LIN {X 99.425,Y -44.827,Z -45.204,A -90.000,B 90.000,C 0.000} C_DIS
LIN {X 99.466,Y -44.816,Z -45.164,A -90.000,B 90.000,C 0.000} C_DIS
LIN {X 99.493,Y -44.805,Z -45.135,A -90.000,B 90.000,C 0.000} C_DIS
LIN {X 99.508,Y -44.792,Z -45.118,A -90.000,B 90.000,C 0.000} C_DIS
LIN {X 99.515,Y -44.777,Z -45.107,A -90.000,B 90.000,C 0.000} C_DIS
LIN {X 99.516,Y -44.768,Z -45.104,A -90.000,B 90.000,C 0.000} C_DIS
LIN {X 99.507,Y -44.687,Z -45.089,A -90.000,B 90.000,C 0.000} C_DIS
LIN {X 99.509,Y -44.621,Z -45.070,A -90.000,B 90.000,C 0.000} C_DIS
LIN {X 99.519,Y -44.564,Z -45.046,A -90.000,B 90.000,C 0.000} C_DIS
LIN {X 99.538,Y -44.495,Z -45.011,A -90.000,B 90.000,C 0.000} C_DIS
LIN {X 99.570,Y -44.412,Z -44.962,A -90.000,B 90.000,C 0.000} C_DIS
LIN {X 99.618,Y -44.314,Z -44.895,A -90.000,B 90.000,C 0.000} C_DIS
LIN {X 99.683,Y -44.199,Z -44.808,A -90.000,B 90.000,C 0.000} C_DIS
LIN {X 99.768,Y -44.065,Z -44.699,A -90.000,B 90.000,C 0.000} C_DIS
LIN {X 99.877,Y -43.910,Z -44.564,A -90.000,B 90.000,C 0.000} C_DIS
LIN {X 100.012,Y -43.731,Z -44.402,A -90.000,B 90.000,C 0.000} C_DIS
LIN {X 100.175,Y -43.526,Z -44.208,A -90.000,B 90.000,C 0.000} C_DIS
LIN {X 100.317,Y -43.354,Z -44.041,A -90.000,B 90.000,C 0.000} C_DIS
LIN {X 100.597,Y -43.062,Z -43.718,A -90.000,B 90.000,C 0.000} C_DIS
LIN {X 100.862,Y -42.817,Z -43.416,A -90.000,B 90.000,C 0.000} C_DIS
LIN {X 101.165,Y -37.308,Z -43.072,A -90.000,B 90.000,C 0.000} C_DIS
LIN {X 101.207,Y -37.308,Z -43.025,A -90.000,B 90.000,C 0.000} C_DIS
LIN {X 101.288,Y -42.488,Z -42.934,A -90.000,B 90.000,C 0.000} C_DIS
LIN {X 101.299,Y -42.484,Z -42.922,A -90.000,B 90.000,C 0.000} C_DIS
LIN {X 101.301,Y -42.492,Z -42.920,A -90.000,B 90.000,C 0.000} C_DIS
LIN {X 101.311,Y -42.494,Z -42.909,A -90.000,B 90.000,C 0.000} C_DIS
LIN {X 101.393,Y -37.308,Z -42.819,A -90.000,B 90.000,C 0.000} C_DIS
LIN {X 101.467,Y -37.311,Z -42.737,A -90.000,B 90.000,C 0.000} C_DIS
LIN {X 101.519,Y -37.308,Z -42.679,A -90.000,B 90.000,C 0.000} C_DIS
LIN {X 101.519,Y -60.000,Z -42.679,A -90.000,B 90.000,C 0.000} C_DIS
LIN {X 91.034,Y -60.000,Z -118.889,A -90.000,B 90.000,C 0.000} C_DIS
LIN {X 91.034,Y -37.308,Z -118.889,A -90.000,B 90.000,C 0.000} C_DIS
LIN {X 91.028,Y -37.310,Z -119.075,A -90.000,B 90.000,C 0.000} C_DIS
LIN {X 91.024,Y -37.317,Z -119.386,A -90.000,B 90.000,C 0.000} C_DIS
LIN {X 91.058,Y -37.308,Z -120.562,A -90.000,B 90.000,C 0.000} C_DIS
LIN {X 91.058,Y -60.000,Z -120.562,A -90.000,B 90.000,C 0.000} C_DIS
LIN {X 18.246,Y -60.000,Z -172.708,A -90.000,B 90.000,C 0.000} C_DIS
LIN {X 18.246,Y -37.308,Z -172.708,A -90.000,B 90.000,C 0.000} C_DIS
LIN {X 18.676,Y -37.337,Z -172.279,A -90.000,B 90.000,C 0.000} C_DIS
LIN {X 19.234,Y -37.370,Z -171.709,A -90.000,B 90.000,C 0.000} C_DIS
LIN {X 19.511,Y -37.385,Z -171.418,A -90.000,B 90.000,C 0.000} C_DIS
LIN {X 20.129,Y -37.438,Z -170.757,A -90.000,B 90.000,C 0.000} C_DIS
LIN {X 20.879,Y -37.487,Z -169.898,A -90.000,B 90.000,C 0.000} C_DIS
LIN {X 21.061,Y -37.497,Z -169.689,A -90.000,B 90.000,C 0.000} C_DIS
LIN {X 21.262,Y -37.507,Z -169.454,A -90.000,B 90.000,C 0.000} C_DIS
LIN {X 21.665,Y -37.542,Z -168.973,A -90.000,B 90.000,C 0.000} C_DIS
LIN {X 21.886,Y -37.558,Z -168.693,A -90.000,B 90.000,C 0.000} C_DIS
LIN {X 22.441,Y -37.593,Z -167.976,A -90.000,B 90.000,C 0.000} C_DIS
LIN {X 22.927,Y -37.634,Z -167.341,A -90.000,B 90.000,C 0.000} C_DIS
LIN {X 23.381,Y -37.667,Z -166.718,A -90.000,B 90.000,C 0.000} C_DIS
LIN {X 23.591,Y -37.681,Z -166.424,A -90.000,B 90.000,C 0.000} C_DIS
LIN {X 23.790,Y -37.709,Z -166.136,A -90.000,B 90.000,C 0.000} C_DIS
LIN {X 23.902,Y -37.722,Z -165.976,A -90.000,B 90.000,C 0.000} C_DIS
LIN {X 24.323,Y -37.756,Z -165.386,A -90.000,B 90.000,C 0.000} C_DIS
LIN {X 24.729,Y -37.786,Z -164.795,A -90.000,B 90.000,C 0.000} C_DIS
LIN {X 25.418,Y -37.885,Z -163.750,A -90.000,B 90.000,C 0.000} C_DIS
LIN {X 25.616,Y -37.899,Z -163.459,A -90.000,B 90.000,C 0.000} C_DIS
LIN {X 25.783,Y -37.929,Z -163.201,A -90.000,B 90.000,C 0.000} C_DIS
LIN {X 26.867,Y -38.118,Z -161.513,A -90.000,B 90.000,C 0.000} C_DIS
LIN {X 26.926,Y -38.131,Z -161.421,A -90.000,B 90.000,C 0.000} C_DIS
LIN {X 27.075,Y -38.162,Z -161.189,A -90.000,B 90.000,C 0.000} C_DIS
LIN {X 27.785,Y -38.314,Z -160.034,A -90.000,B 90.000,C 0.000} C_DIS
LIN {X 28.223,Y -38.430,Z -159.320,A -90.000,B 90.000,C 0.000} C_DIS
LIN {X 28.758,Y -38.583,Z -158.366,A -90.000,B 90.000,C 0.000} C_DIS
LIN {X 29.089,Y -38.675,Z -157.778,A -90.000,B 90.000,C 0.000} C_DIS
LIN {X 28.763,Y -38.667,Z -157.817,A -90.000,B 90.000,C 0.000} C_DIS
LIN {X 28.657,Y -38.665,Z -157.825,A -90.000,B 90.000,C 0.000} C_DIS
LIN {X 28.540,Y -38.663,Z -157.832,A -90.000,B 90.000,C 0.000} C_DIS
LIN {X 28.360,Y -38.661,Z -157.834,A -90.000,B 90.000,C 0.000} C_DIS
LIN {X 28.193,Y -38.664,Z -157.832,A -90.000,B 90.000,C 0.000} C_DIS
LIN {X 27.973,Y -38.669,Z -157.816,A -90.000,B 90.000,C 0.000} C_DIS
LIN {X 27.602,Y -38.679,Z -157.774,A -90.000,B 90.000,C 0.000} C_DIS
LIN {X 27.471,Y -38.683,Z -157.755,A -90.000,B 90.000,C 0.000} C_DIS
LIN {X 27.348,Y -38.686,Z -157.733,A -90.000,B 90.000,C 0.000} C_DIS
LIN {X 27.168,Y -38.691,Z -157.696,A -90.000,B 90.000,C 0.000} C_DIS
LIN {X 26.963,Y -38.699,Z -157.642,A -90.000,B 90.000,C 0.000} C_DIS
LIN {X 26.817,Y -38.705,Z -157.597,A -90.000,B 90.000,C 0.000} C_DIS
LIN {X 26.706,Y -38.710,Z -157.559,A -90.000,B 90.000,C 0.000} C_DIS
LIN {X 26.470,Y -38.713,Z -157.462,A -90.000,B 90.000,C 0.000} C_DIS
LIN {X 26.304,Y -38.715,Z -157.392,A -90.000,B 90.000,C 0.000} C_DIS
LIN {X 26.199,Y -38.718,Z -157.343,A -90.000,B 90.000,C 0.000} C_DIS
LIN {X 26.036,Y -38.724,Z -157.251,A -90.000,B 90.000,C 0.000} C_DIS
LIN {X 25.598,Y -38.746,Z -156.984,A -90.000,B 90.000,C 0.000} C_DIS
LIN {X 25.482,Y -38.751,Z -156.901,A -90.000,B 90.000,C 0.000} C_DIS
LIN {X 25.247,Y -38.759,Z -156.714,A -90.000,B 90.000,C 0.000} C_DIS
LIN {X 25.138,Y -38.762,Z -156.620,A -90.000,B 90.000,C 0.000} C_DIS
LIN {X 25.035,Y -38.762,Z -156.525,A -90.000,B 90.000,C 0.000} C_DIS
LIN {X 24.917,Y -38.757,Z -156.404,A -90.000,B 90.000,C 0.000} C_DIS
LIN {X 24.794,Y -38.750,Z -156.269,A -90.000,B 90.000,C 0.000} C_DIS
LIN {X 24.611,Y -38.747,Z -156.042,A -90.000,B 90.000,C 0.000} C_DIS
LIN {X 24.050,Y -38.739,Z -155.340,A -90.000,B 90.000,C 0.000} C_DIS
LIN {X 23.907,Y -38.734,Z -155.160,A -90.000,B 90.000,C 0.000} C_DIS
LIN {X 23.791,Y -38.721,Z -155.008,A -90.000,B 90.000,C 0.000} C_DIS
LIN {X 23.677,Y -38.702,Z -154.847,A -90.000,B 90.000,C 0.000} C_DIS
LIN {X 23.524,Y -38.677,Z -154.617,A -90.000,B 90.000,C 0.000} C_DIS
LIN {X 23.421,Y -38.661,Z -154.444,A -90.000,B 90.000,C 0.000} C_DIS
LIN {X 23.386,Y -38.655,Z -154.380,A -90.000,B 90.000,C 0.000} C_DIS
LIN {X 23.328,Y -38.647,Z -154.260,A -90.000,B 90.000,C 0.000} C_DIS
LIN {X 23.170,Y -38.626,Z -153.901,A -90.000,B 90.000,C 0.000} C_DIS
LIN {X 23.071,Y -38.615,Z -153.627,A -90.000,B 90.000,C 0.000} C_DIS
LIN {X 23.025,Y -38.608,Z -153.480,A -90.000,B 90.000,C 0.000} C_DIS
LIN {X 23.006,Y -38.602,Z -153.415,A -90.000,B 90.000,C 0.000} C_DIS
LIN {X 22.974,Y -38.590,Z -153.292,A -90.000,B 90.000,C 0.000} C_DIS
LIN {X 22.949,Y -38.580,Z -153.182,A -90.000,B 90.000,C 0.000} C_DIS
LIN {X 22.929,Y -38.570,Z -153.079,A -90.000,B 90.000,C 0.000} C_DIS
LIN {X 22.906,Y -38.558,Z -152.910,A -90.000,B 90.000,C 0.000} C_DIS
LIN {X 22.877,Y -38.535,Z -152.666,A -90.000,B 90.000,C 0.000} C_DIS
LIN {X 22.866,Y -38.520,Z -152.493,A -90.000,B 90.000,C 0.000} C_DIS
LIN {X 22.858,Y -38.505,Z -152.287,A -90.000,B 90.000,C 0.000} C_DIS
LIN {X 22.857,Y -38.492,Z -152.102,A -90.000,B 90.000,C 0.000} C_DIS
LIN {X 22.860,Y -38.479,Z -151.897,A -90.000,B 90.000,C 0.000} C_DIS
LIN {X 22.879,Y -38.466,Z -151.654,A -90.000,B 90.000,C 0.000} C_DIS
LIN {X 22.890,Y -38.460,Z -151.561,A -90.000,B 90.000,C 0.000} C_DIS
LIN {X 22.930,Y -38.448,Z -151.318,A -90.000,B 90.000,C 0.000} C_DIS
LIN {X 22.962,Y -38.439,Z -151.169,A -90.000,B 90.000,C 0.000} C_DIS
LIN {X 23.121,Y -38.404,Z -150.496,A -90.000,B 90.000,C 0.000} C_DIS
LIN {X 23.299,Y -38.353,Z -149.757,A -90.000,B 90.000,C 0.000} C_DIS
LIN {X 23.377,Y -38.318,Z -149.455,A -90.000,B 90.000,C 0.000} C_DIS
LIN {X 23.475,Y -38.278,Z -149.098,A -90.000,B 90.000,C 0.000} C_DIS
LIN {X 22.762,Y -38.124,Z -149.465,A -90.000,B 90.000,C 0.000} C_DIS
LIN {X 22.308,Y -38.024,Z -149.687,A -90.000,B 90.000,C 0.000} C_DIS
LIN {X 21.806,Y -37.911,Z -149.923,A -90.000,B 90.000,C 0.000} C_DIS
LIN {X 21.521,Y -37.843,Z -150.045,A -90.000,B 90.000,C 0.000} C_DIS
LIN {X 21.069,Y -37.732,Z -150.227,A -90.000,B 90.000,C 0.000} C_DIS
LIN {X 20.845,Y -37.674,Z -150.314,A -90.000,B 90.000,C 0.000} C_DIS
LIN {X 20.751,Y -37.647,Z -150.349,A -90.000,B 90.000,C 0.000} C_DIS
LIN {X 20.361,Y -37.529,Z -150.492,A -90.000,B 90.000,C 0.000} C_DIS
LIN {X 20.188,Y -37.475,Z -150.553,A -90.000,B 90.000,C 0.000} C_DIS
LIN {X 19.812,Y -37.357,Z -150.680,A -90.000,B 90.000,C 0.000} C_DIS
LIN {X 19.659,Y -37.308,Z -150.727,A -90.000,B 90.000,C 0.000} C_DIS
LIN {X 19.659,Y -60.000,Z -150.727,A -90.000,B 90.000,C 0.000} C_DIS
LIN {X 22.617,Y -60.000,Z -164.416,A -90.000,B 90.000,C 0.000} C_DIS
LIN {X 22.617,Y -37.308,Z -164.416,A -90.000,B 90.000,C 0.000} C_DIS
LIN {X 22.733,Y -37.343,Z -164.245,A -90.000,B 90.000,C 0.000} C_DIS
LIN {X 23.104,Y -37.453,Z -163.677,A -90.000,B 90.000,C 0.000} C_DIS
LIN {X 23.691,Y -37.627,Z -162.765,A -90.000,B 90.000,C 0.000} C_DIS
LIN {X 23.962,Y -37.712,Z -162.351,A -90.000,B 90.000,C 0.000} C_DIS
LIN {X 24.575,Y -37.908,Z -161.385,A -90.000,B 90.000,C 0.000} C_DIS
LIN {X 25.260,Y -38.149,Z -160.314,A -90.000,B 90.000,C 0.000} C_DIS
LIN {X 25.375,Y -38.189,Z -160.136,A -90.000,B 90.000,C 0.000} C_DIS
LIN {X 25.866,Y -38.354,Z -159.341,A -90.000,B 90.000,C 0.000} C_DIS
LIN {X 25.505,Y -38.359,Z -159.191,A -90.000,B 90.000,C 0.000} C_DIS
LIN {X 25.293,Y -38.363,Z -159.090,A -90.000,B 90.000,C 0.000} C_DIS
LIN {X 25.088,Y -38.371,Z -158.977,A -90.000,B 90.000,C 0.000} C_DIS
LIN {X 24.998,Y -38.375,Z -158.925,A -90.000,B 90.000,C 0.000} C_DIS
LIN {X 24.767,Y -38.384,Z -158.783,A -90.000,B 90.000,C 0.000} C_DIS
LIN {X 24.591,Y -38.384,Z -158.674,A -90.000,B 90.000,C 0.000} C_DIS
LIN {X 24.446,Y -38.384,Z -158.578,A -90.000,B 90.000,C 0.000} C_DIS
LIN {X 24.331,Y -38.386,Z -158.495,A -90.000,B 90.000,C 0.000} C_DIS
LIN {X 24.251,Y -38.388,Z -158.435,A -90.000,B 90.000,C 0.000} C_DIS
LIN {X 24.016,Y -38.394,Z -158.248,A -90.000,B 90.000,C 0.000} C_DIS
LIN {X 23.824,Y -38.401,Z -158.084,A -90.000,B 90.000,C 0.000} C_DIS
LIN {X 23.677,Y -38.403,Z -157.949,A -90.000,B 90.000,C 0.000} C_DIS
LIN {X 23.542,Y -38.396,Z -157.812,A -90.000,B 90.000,C 0.000} C_DIS
LIN {X 23.436,Y -38.389,Z -157.699,A -90.000,B 90.000,C 0.000} C_DIS
LIN {X 23.308,Y -38.381,Z -157.555,A -90.000,B 90.000,C 0.000} C_DIS
LIN {X 22.995,Y -38.364,Z -157.164,A -90.000,B 90.000,C 0.000} C_DIS
LIN {X 22.933,Y -38.361,Z -157.086,A -90.000,B 90.000,C 0.000} C_DIS
LIN {X 22.850,Y -38.356,Z -156.982,A -90.000,B 90.000,C 0.000} C_DIS
LIN {X 22.614,Y -38.352,Z -156.685,A -90.000,B 90.000,C 0.000} C_DIS
LIN {X 22.511,Y -38.348,Z -156.555,A -90.000,B 90.000,C 0.000} C_DIS
LIN {X 22.379,Y -38.333,Z -156.386,A -90.000,B 90.000,C 0.000} C_DIS
LIN {X 22.216,Y -38.305,Z -156.169,A -90.000,B 90.000,C 0.000} C_DIS
LIN {X 22.071,Y -38.279,Z -155.962,A -90.000,B 90.000,C 0.000} C_DIS
LIN {X 21.887,Y -38.248,Z -155.683,A -90.000,B 90.000,C 0.000} C_DIS
LIN {X 21.768,Y -38.229,Z -155.484,A -90.000,B 90.000,C 0.000} C_DIS
LIN {X 21.691,Y -38.217,Z -155.345,A -90.000,B 90.000,C 0.000} C_DIS
LIN {X 21.617,Y -38.206,Z -155.200,A -90.000,B 90.000,C 0.000} C_DIS
LIN {X 21.556,Y -38.197,Z -155.070,A -90.000,B 90.000,C 0.000} C_DIS
LIN {X 21.488,Y -38.185,Z -154.914,A -90.000,B 90.000,C 0.000} C_DIS
LIN {X 21.411,Y -38.163,Z -154.732,A -90.000,B 90.000,C 0.000} C_DIS
LIN {X 21.349,Y -38.144,Z -154.572,A -90.000,B 90.000,C 0.000} C_DIS
LIN {X 21.232,Y -38.110,Z -154.231,A -90.000,B 90.000,C 0.000} C_DIS
LIN {X 21.148,Y -38.084,Z -153.946,A -90.000,B 90.000,C 0.000} C_DIS
LIN {X 21.104,Y -38.067,Z -153.773,A -90.000,B 90.000,C 0.000} C_DIS
LIN {X 21.062,Y -38.048,Z -153.578,A -90.000,B 90.000,C 0.000} C_DIS
LIN {X 21.032,Y -38.034,Z -153.418,A -90.000,B 90.000,C 0.000} C_DIS
LIN {X 20.994,Y -38.014,Z -153.140,A -90.000,B 90.000,C 0.000} C_DIS
LIN {X 20.968,Y -37.998,Z -152.925,A -90.000,B 90.000,C 0.000} C_DIS
LIN {X 20.955,Y -37.988,Z -152.775,A -90.000,B 90.000,C 0.000} C_DIS
LIN {X 20.945,Y -37.976,Z -152.609,A -90.000,B 90.000,C 0.000} C_DIS
LIN {X 20.936,Y -37.959,Z -152.359,A -90.000,B 90.000,C 0.000} C_DIS
LIN {X 20.612,Y -37.866,Z -152.471,A -90.000,B 90.000,C 0.000} C_DIS
LIN {X 20.258,Y -37.764,Z -152.587,A -90.000,B 90.000,C 0.000} C_DIS
LIN {X 20.104,Y -37.719,Z -152.633,A -90.000,B 90.000,C 0.000} C_DIS
LIN {X 19.527,Y -37.545,Z -152.708,A -90.000,B 90.000,C 0.000} C_DIS
LIN {X 19.410,Y -37.509,Z -152.701,A -90.000,B 90.000,C 0.000} C_DIS
LIN {X 19.315,Y -37.479,Z -152.689,A -90.000,B 90.000,C 0.000} C_DIS
LIN {X 19.266,Y -37.463,Z -152.682,A -90.000,B 90.000,C 0.000} C_DIS
LIN {X 19.149,Y -37.425,Z -152.657,A -90.000,B 90.000,C 0.000} C_DIS
LIN {X 19.091,Y -37.406,Z -152.642,A -90.000,B 90.000,C 0.000} C_DIS
LIN {X 18.945,Y -37.358,Z -152.594,A -90.000,B 90.000,C 0.000} C_DIS
LIN {X 18.894,Y -37.340,Z -152.574,A -90.000,B 90.000,C 0.000} C_DIS
LIN {X 18.810,Y -37.308,Z -152.537,A -90.000,B 90.000,C 0.000} C_DIS
LIN {X 18.810,Y -60.000,Z -152.537,A -90.000,B 90.000,C 0.000} C_DIS
LIN {X 21.484,Y -60.000,Z -162.510,A -90.000,B 90.000,C 0.000} C_DIS
LIN {X 21.484,Y -37.308,Z -162.510,A -90.000,B 90.000,C 0.000} C_DIS
LIN {X 21.876,Y -37.483,Z -161.895,A -90.000,B 90.000,C 0.000} C_DIS
LIN {X 22.026,Y -37.546,Z -161.659,A -90.000,B 90.000,C 0.000} C_DIS
LIN {X 22.297,Y -37.662,Z -161.243,A -90.000,B 90.000,C 0.000} C_DIS
LIN {X 23.082,Y -37.985,Z -160.008,A -90.000,B 90.000,C 0.000} C_DIS
LIN {X 22.787,Y -37.991,Z -159.774,A -90.000,B 90.000,C 0.000} C_DIS
LIN {X 22.571,Y -37.983,Z -159.586,A -90.000,B 90.000,C 0.000} C_DIS
LIN {X 22.497,Y -37.980,Z -159.520,A -90.000,B 90.000,C 0.000} C_DIS
LIN {X 22.296,Y -37.971,Z -159.329,A -90.000,B 90.000,C 0.000} C_DIS
LIN {X 22.236,Y -37.969,Z -159.269,A -90.000,B 90.000,C 0.000} C_DIS
LIN {X 22.077,Y -37.956,Z -159.103,A -90.000,B 90.000,C 0.000} C_DIS
LIN {X 21.980,Y -37.944,Z -158.996,A -90.000,B 90.000,C 0.000} C_DIS
LIN {X 21.844,Y -37.927,Z -158.840,A -90.000,B 90.000,C 0.000} C_DIS
LIN {X 21.720,Y -37.913,Z -158.684,A -90.000,B 90.000,C 0.000} C_DIS
LIN {X 21.264,Y -37.892,Z -158.113,A -90.000,B 90.000,C 0.000} C_DIS
LIN {X 21.115,Y -37.884,Z -157.924,A -90.000,B 90.000,C 0.000} C_DIS
LIN {X 20.990,Y -37.866,Z -157.761,A -90.000,B 90.000,C 0.000} C_DIS
LIN {X 20.835,Y -37.840,Z -157.559,A -90.000,B 90.000,C 0.000} C_DIS
LIN {X 20.635,Y -37.803,Z -157.287,A -90.000,B 90.000,C 0.000} C_DIS
LIN {X 20.482,Y -37.779,Z -157.068,A -90.000,B 90.000,C 0.000} C_DIS
LIN {X 20.297,Y -37.751,Z -156.789,A -90.000,B 90.000,C 0.000} C_DIS
LIN {X 20.213,Y -37.739,Z -156.654,A -90.000,B 90.000,C 0.000} C_DIS
LIN {X 20.089,Y -37.722,Z -156.444,A -90.000,B 90.000,C 0.000} C_DIS
LIN {X 19.980,Y -37.709,Z -156.249,A -90.000,B 90.000,C 0.000} C_DIS
LIN {X 19.867,Y -37.686,Z -156.016,A -90.000,B 90.000,C 0.000} C_DIS
LIN {X 19.744,Y -37.658,Z -155.740,A -90.000,B 90.000,C 0.000} C_DIS
LIN {X 19.635,Y -37.632,Z -155.484,A -90.000,B 90.000,C 0.000} C_DIS
LIN {X 19.572,Y -37.617,Z -155.324,A -90.000,B 90.000,C 0.000} C_DIS
LIN {X 19.541,Y -37.610,Z -155.241,A -90.000,B 90.000,C 0.000} C_DIS
LIN {X 19.422,Y -37.583,Z -154.899,A -90.000,B 90.000,C 0.000} C_DIS
LIN {X 19.361,Y -37.570,Z -154.701,A -90.000,B 90.000,C 0.000} C_DIS
LIN {X 19.198,Y -37.517,Z -154.690,A -90.000,B 90.000,C 0.000} C_DIS
LIN {X 19.005,Y -37.454,Z -154.665,A -90.000,B 90.000,C 0.000} C_DIS
LIN {X 18.852,Y -37.405,Z -154.637,A -90.000,B 90.000,C 0.000} C_DIS
LIN {X 18.741,Y -37.370,Z -154.614,A -90.000,B 90.000,C 0.000} C_DIS
LIN {X 18.608,Y -37.327,Z -154.581,A -90.000,B 90.000,C 0.000} C_DIS
LIN {X 18.552,Y -37.308,Z -154.565,A -90.000,B 90.000,C 0.000} C_DIS
LIN {X 18.417,Y -37.265,Z -154.530,A -90.000,B 90.000,C 0.000} C_DIS
LIN {X 18.286,Y -37.220,Z -154.499,A -90.000,B 90.000,C 0.000} C_DIS
LIN {X 18.158,Y -37.176,Z -154.474,A -90.000,B 90.000,C 0.000} C_DIS
LIN {X 18.033,Y -37.133,Z -154.454,A -90.000,B 90.000,C 0.000} C_DIS
LIN {X 17.913,Y -37.092,Z -154.438,A -90.000,B 90.000,C 0.000} C_DIS
LIN {X 17.796,Y -37.052,Z -154.428,A -90.000,B 90.000,C 0.000} C_DIS
LIN {X 17.682,Y -37.013,Z -154.422,A -90.000,B 90.000,C 0.000} C_DIS
LIN {X 17.518,Y -36.957,Z -154.423,A -90.000,B 90.000,C 0.000} C_DIS
LIN {X 17.413,Y -36.921,Z -154.429,A -90.000,B 90.000,C 0.000} C_DIS
LIN {X 17.311,Y -36.887,Z -154.439,A -90.000,B 90.000,C 0.000} C_DIS
LIN {X 17.213,Y -36.854,Z -154.454,A -90.000,B 90.000,C 0.000} C_DIS
LIN {X 17.072,Y -36.807,Z -154.485,A -90.000,B 90.000,C 0.000} C_DIS
LIN {X 16.982,Y -36.777,Z -154.510,A -90.000,B 90.000,C 0.000} C_DIS
LIN {X 16.896,Y -36.748,Z -154.539,A -90.000,B 90.000,C 0.000} C_DIS
LIN {X 16.812,Y -36.721,Z -154.573,A -90.000,B 90.000,C 0.000} C_DIS
LIN {X 16.693,Y -36.682,Z -154.630,A -90.000,B 90.000,C 0.000} C_DIS
LIN {X 16.618,Y -36.657,Z -154.673,A -90.000,B 90.000,C 0.000} C_DIS
LIN {X 16.545,Y -36.634,Z -154.719,A -90.000,B 90.000,C 0.000} C_DIS
LIN {X 16.476,Y -36.611,Z -154.769,A -90.000,B 90.000,C 0.000} C_DIS
LIN {X 16.378,Y -36.580,Z -154.851,A -90.000,B 90.000,C 0.000} C_DIS
LIN {X 16.316,Y -36.560,Z -154.909,A -90.000,B 90.000,C 0.000} C_DIS
LIN {X 16.229,Y -36.530,Z -155.003,A -90.000,B 90.000,C 0.000} C_DIS
LIN {X 16.175,Y -36.511,Z -155.069,A -90.000,B 90.000,C 0.000} C_DIS
LIN {X 16.099,Y -36.483,Z -155.174,A -90.000,B 90.000,C 0.000} C_DIS
LIN {X 16.007,Y -36.446,Z -155.323,A -90.000,B 90.000,C 0.000} C_DIS
LIN {X 15.965,Y -36.428,Z -155.402,A -90.000,B 90.000,C 0.000} C_DIS
LIN {X 15.891,Y -36.387,Z -155.567,A -90.000,B 90.000,C 0.000} C_DIS
LIN {X 15.826,Y -36.349,Z -155.742,A -90.000,B 90.000,C 0.000} C_DIS
LIN {X 15.798,Y -36.331,Z -155.833,A -90.000,B 90.000,C 0.000} C_DIS
LIN {X 15.750,Y -36.297,Z -156.020,A -90.000,B 90.000,C 0.000} C_DIS
LIN {X 15.712,Y -36.266,Z -156.215,A -90.000,B 90.000,C 0.000} C_DIS
LIN {X 15.683,Y -36.238,Z -156.416,A -90.000,B 90.000,C 0.000} C_DIS
LIN {X 15.664,Y -36.214,Z -156.624,A -90.000,B 90.000,C 0.000} C_DIS
LIN {X 15.655,Y -36.192,Z -156.837,A -90.000,B 90.000,C 0.000} C_DIS
LIN {X 15.654,Y -36.168,Z -157.055,A -90.000,B 90.000,C 0.000} C_DIS
LIN {X 15.663,Y -36.139,Z -157.276,A -90.000,B 90.000,C 0.000} C_DIS
LIN {X 15.670,Y -36.125,Z -157.388,A -90.000,B 90.000,C 0.000} C_DIS
LIN {X 15.691,Y -36.100,Z -157.613,A -90.000,B 90.000,C 0.000} C_DIS
LIN {X 15.721,Y -36.078,Z -157.841,A -90.000,B 90.000,C 0.000} C_DIS
LIN {X 15.758,Y -36.064,Z -158.069,A -90.000,B 90.000,C 0.000} C_DIS
LIN {X 15.803,Y -36.055,Z -158.298,A -90.000,B 90.000,C 0.000} C_DIS
LIN {X 15.856,Y -36.047,Z -158.527,A -90.000,B 90.000,C 0.000} C_DIS
LIN {X 15.916,Y -36.040,Z -158.754,A -90.000,B 90.000,C 0.000} C_DIS
LIN {X 15.982,Y -36.035,Z -158.980,A -90.000,B 90.000,C 0.000} C_DIS
LIN {X 16.056,Y -36.034,Z -159.203,A -90.000,B 90.000,C 0.000} C_DIS
LIN {X 16.135,Y -36.036,Z -159.423,A -90.000,B 90.000,C 0.000} C_DIS
LIN {X 16.221,Y -36.040,Z -159.638,A -90.000,B 90.000,C 0.000} C_DIS
LIN {X 16.313,Y -36.046,Z -159.849,A -90.000,B 90.000,C 0.000} C_DIS
LIN {X 16.411,Y -36.054,Z -160.054,A -90.000,B 90.000,C 0.000} C_DIS
LIN {X 16.514,Y -36.068,Z -160.253,A -90.000,B 90.000,C 0.000} C_DIS
LIN {X 16.567,Y -36.077,Z -160.350,A -90.000,B 90.000,C 0.000} C_DIS
LIN {X 16.678,Y -36.095,Z -160.538,A -90.000,B 90.000,C 0.000} C_DIS
LIN {X 16.793,Y -36.117,Z -160.717,A -90.000,B 90.000,C 0.000} C_DIS
LIN {X 16.913,Y -36.142,Z -160.888,A -90.000,B 90.000,C 0.000} C_DIS
LIN {X 17.038,Y -36.169,Z -161.049,A -90.000,B 90.000,C 0.000} C_DIS
LIN {X 17.166,Y -36.199,Z -161.199,A -90.000,B 90.000,C 0.000} C_DIS
LIN {X 17.298,Y -36.226,Z -161.338,A -90.000,B 90.000,C 0.000} C_DIS
LIN {X 17.433,Y -36.257,Z -161.465,A -90.000,B 90.000,C 0.000} C_DIS
LIN {X 17.572,Y -36.291,Z -161.580,A -90.000,B 90.000,C 0.000} C_DIS
LIN {X 17.714,Y -36.327,Z -161.680,A -90.000,B 90.000,C 0.000} C_DIS
LIN {X 17.858,Y -36.367,Z -161.767,A -90.000,B 90.000,C 0.000} C_DIS
LIN {X 18.006,Y -36.409,Z -161.839,A -90.000,B 90.000,C 0.000} C_DIS
LIN {X 18.117,Y -36.442,Z -161.882,A -90.000,B 90.000,C 0.000} C_DIS
LIN {X 18.230,Y -36.477,Z -161.916,A -90.000,B 90.000,C 0.000} C_DIS
LIN {X 18.306,Y -36.501,Z -161.934,A -90.000,B 90.000,C 0.000} C_DIS
LIN {X 18.382,Y -36.525,Z -161.947,A -90.000,B 90.000,C 0.000} C_DIS
LIN {X 18.497,Y -36.563,Z -161.959,A -90.000,B 90.000,C 0.000} C_DIS
LIN {X 18.575,Y -36.590,Z -161.961,A -90.000,B 90.000,C 0.000} C_DIS
LIN {X 18.652,Y -36.617,Z -161.958,A -90.000,B 90.000,C 0.000} C_DIS
LIN {X 18.769,Y -36.658,Z -161.945,A -90.000,B 90.000,C 0.000} C_DIS
LIN {X 18.847,Y -36.686,Z -161.931,A -90.000,B 90.000,C 0.000} C_DIS
LIN {X 18.926,Y -36.715,Z -161.911,A -90.000,B 90.000,C 0.000} C_DIS
LIN {X 19.044,Y -36.758,Z -161.872,A -90.000,B 90.000,C 0.000} C_DIS
LIN {X 19.162,Y -36.803,Z -161.822,A -90.000,B 90.000,C 0.000} C_DIS
LIN {X 19.280,Y -36.849,Z -161.759,A -90.000,B 90.000,C 0.000} C_DIS
LIN {X 19.359,Y -36.881,Z -161.710,A -90.000,B 90.000,C 0.000} C_DIS
LIN {X 19.438,Y -36.914,Z -161.656,A -90.000,B 90.000,C 0.000} C_DIS
LIN {X 19.557,Y -36.965,Z -161.564,A -90.000,B 90.000,C 0.000} C_DIS
LIN {X 19.675,Y -37.017,Z -161.459,A -90.000,B 90.000,C 0.000} C_DIS
LIN {X 19.793,Y -37.072,Z -161.341,A -90.000,B 90.000,C 0.000} C_DIS
LIN {X 19.911,Y -37.129,Z -161.208,A -90.000,B 90.000,C 0.000} C_DIS
LIN {X 20.028,Y -37.187,Z -161.062,A -90.000,B 90.000,C 0.000} C_DIS
LIN {X 20.106,Y -37.227,Z -160.957,A -90.000,B 90.000,C 0.000} C_DIS
LIN {X 20.183,Y -37.267,Z -160.845,A -90.000,B 90.000,C 0.000} C_DIS
LIN {X 20.260,Y -37.308,Z -160.726,A -90.000,B 90.000,C 0.000} C_DIS
LIN {X 20.369,Y -37.366,Z -160.555,A -90.000,B 90.000,C 0.000} C_DIS
LIN {X 20.539,Y -37.447,Z -160.291,A -90.000,B 90.000,C 0.000} C_DIS
LIN {X 20.399,Y -37.429,Z -160.130,A -90.000,B 90.000,C 0.000} C_DIS
LIN {X 20.212,Y -37.409,Z -159.898,A -90.000,B 90.000,C 0.000} C_DIS
LIN {X 19.728,Y -37.358,Z -159.279,A -90.000,B 90.000,C 0.000} C_DIS
LIN {X 19.584,Y -37.337,Z -159.090,A -90.000,B 90.000,C 0.000} C_DIS
LIN {X 19.416,Y -37.308,Z -158.870,A -90.000,B 90.000,C 0.000} C_DIS
LIN {X 19.416,Y -60.000,Z -158.870,A -90.000,B 90.000,C 0.000} C_DIS
LIN {X -17.979,Y -60.000,Z -204.513,A -90.000,B 90.000,C 0.000} C_DIS
LIN {X -17.979,Y -37.308,Z -204.513,A -90.000,B 90.000,C 0.000} C_DIS
LIN {X -17.744,Y -37.310,Z -204.358,A -90.000,B 90.000,C 0.000} C_DIS
LIN {X -17.409,Y -37.320,Z -204.135,A -90.000,B 90.000,C 0.000} C_DIS
LIN {X -16.506,Y -37.350,Z -203.542,A -90.000,B 90.000,C 0.000} C_DIS
LIN {X -16.323,Y -37.355,Z -203.419,A -90.000,B 90.000,C 0.000} C_DIS
LIN {X -14.126,Y -37.380,Z -201.881,A -90.000,B 90.000,C 0.000} C_DIS
LIN {X -12.515,Y -37.430,Z -200.733,A -90.000,B 90.000,C 0.000} C_DIS
LIN {X -11.622,Y -37.438,Z -200.059,A -90.000,B 90.000,C 0.000} C_DIS
LIN {X -10.479,Y -37.445,Z -199.199,A -90.000,B 90.000,C 0.000} C_DIS
LIN {X -8.852,Y -37.480,Z -197.959,A -90.000,B 90.000,C 0.000} C_DIS
LIN {X -6.807,Y -37.483,Z -196.303,A -90.000,B 90.000,C 0.000} C_DIS
LIN {X -5.675,Y -37.503,Z -195.382,A -90.000,B 90.000,C 0.000} C_DIS
LIN {X -5.363,Y -37.507,Z -195.128,A -90.000,B 90.000,C 0.000} C_DIS
LIN {X -3.165,Y -37.487,Z -193.219,A -90.000,B 90.000,C 0.000} C_DIS
LIN {X -2.606,Y -37.486,Z -192.733,A -90.000,B 90.000,C 0.000} C_DIS
LIN {X -1.907,Y -37.489,Z -192.136,A -90.000,B 90.000,C 0.000} C_DIS
LIN {X -1.355,Y -37.484,Z -191.648,A -90.000,B 90.000,C 0.000} C_DIS
LIN {X -0.812,Y -37.470,Z -191.143,A -90.000,B 90.000,C 0.000} C_DIS
LIN {X 0.673,Y -37.448,Z -189.749,A -90.000,B 90.000,C 0.000} C_DIS
LIN {X 1.666,Y -37.427,Z -188.823,A -90.000,B 90.000,C 0.000} C_DIS
LIN {X 1.924,Y -37.424,Z -188.587,A -90.000,B 90.000,C 0.000} C_DIS
LIN {X 2.619,Y -37.401,Z -187.917,A -90.000,B 90.000,C 0.000} C_DIS
LIN {X 4.131,Y -37.372,Z -186.440,A -90.000,B 90.000,C 0.000} C_DIS
LIN {X 5.120,Y -37.344,Z -185.483,A -90.000,B 90.000,C 0.000} C_DIS
LIN {X 6.009,Y -37.315,Z -184.612,A -90.000,B 90.000,C 0.000} C_DIS
LIN {X 6.346,Y -37.308,Z -184.277,A -90.000,B 90.000,C 0.000} C_DIS
LIN {X 6.346,Y -60.000,Z -184.277,A -90.000,B 90.000,C 0.000} C_DIS
LIN {X -35.487,Y -60.000,Z -96.281,A -90.000,B 90.000,C 0.000} C_DIS
LIN {X -35.487,Y -37.308,Z -96.281,A -90.000,B 90.000,C 0.000} C_DIS
LIN {X -35.355,Y -37.473,Z -95.669,A -90.000,B 90.000,C 0.000} C_DIS
LIN {X -35.299,Y -37.539,Z -95.419,A -90.000,B 90.000,C 0.000} C_DIS
LIN {X -35.280,Y -37.573,Z -95.284,A -90.000,B 90.000,C 0.000} C_DIS
LIN {X -35.250,Y -37.617,Z -95.079,A -90.000,B 90.000,C 0.000} C_DIS
LIN {X -35.224,Y -37.658,Z -94.884,A -90.000,B 90.000,C 0.000} C_DIS
LIN {X -35.157,Y -37.756,Z -94.429,A -90.000,B 90.000,C 0.000} C_DIS
LIN {X -35.110,Y -37.820,Z -94.133,A -90.000,B 90.000,C 0.000} C_DIS
LIN {X -35.034,Y -37.912,Z -93.725,A -90.000,B 90.000,C 0.000} C_DIS
LIN {X -35.018,Y -37.930,Z -93.648,A -90.000,B 90.000,C 0.000} C_DIS
LIN {X -34.929,Y -38.020,Z -93.261,A -90.000,B 90.000,C 0.000} C_DIS
LIN {X -34.800,Y -38.139,Z -92.757,A -90.000,B 90.000,C 0.000} C_DIS
LIN {X -34.696,Y -38.210,Z -92.368,A -90.000,B 90.000,C 0.000} C_DIS
LIN {X -34.550,Y -38.318,Z -91.745,A -90.000,B 90.000,C 0.000} C_DIS
LIN {X -34.444,Y -38.391,Z -91.330,A -90.000,B 90.000,C 0.000} C_DIS
LIN {X -34.381,Y -38.431,Z -91.120,A -90.000,B 90.000,C 0.000} C_DIS
LIN {X -34.365,Y -38.440,Z -91.068,A -90.000,B 90.000,C 0.000} C_DIS
LIN {X -34.250,Y -38.518,Z -90.637,A -90.000,B 90.000,C 0.000} C_DIS
LIN {X -34.191,Y -38.542,Z -90.430,A -90.000,B 90.000,C 0.000} C_DIS
LIN {X -34.082,Y -38.582,Z -90.074,A -90.000,B 90.000,C 0.000} C_DIS
LIN {X -34.040,Y -38.595,Z -89.940,A -90.000,B 90.000,C 0.000} C_DIS
LIN {X -34.026,Y -38.605,Z -89.760,A -90.000,B 90.000,C 0.000} C_DIS
LIN {X -33.987,Y -38.624,Z -89.463,A -90.000,B 90.000,C 0.000} C_DIS
LIN {X -33.966,Y -38.633,Z -89.340,A -90.000,B 90.000,C 0.000} C_DIS
LIN {X -33.781,Y -38.705,Z -88.408,A -90.000,B 90.000,C 0.000} C_DIS
LIN {X -33.711,Y -38.733,Z -88.060,A -90.000,B 90.000,C 0.000} C_DIS
LIN {X -33.677,Y -38.739,Z -87.893,A -90.000,B 90.000,C 0.000} C_DIS
LIN {X -33.491,Y -38.742,Z -87.055,A -90.000,B 90.000,C 0.000} C_DIS
LIN {X -33.452,Y -38.743,Z -86.877,A -90.000,B 90.000,C 0.000} C_DIS
LIN {X -33.409,Y -38.744,Z -86.697,A -90.000,B 90.000,C 0.000} C_DIS
LIN {X -33.370,Y -38.746,Z -86.555,A -90.000,B 90.000,C 0.000} C_DIS
LIN {X -33.327,Y -38.748,Z -86.420,A -90.000,B 90.000,C 0.000} C_DIS
LIN {X -33.290,Y -38.750,Z -86.313,A -90.000,B 90.000,C 0.000} C_DIS
LIN {X -33.213,Y -38.756,Z -86.120,A -90.000,B 90.000,C 0.000} C_DIS
LIN {X -33.166,Y -38.760,Z -86.013,A -90.000,B 90.000,C 0.000} C_DIS
LIN {X -33.088,Y -38.767,Z -85.853,A -90.000,B 90.000,C 0.000} C_DIS
LIN {X -33.027,Y -38.772,Z -85.739,A -90.000,B 90.000,C 0.000} C_DIS
LIN {X -32.941,Y -38.772,Z -85.581,A -90.000,B 90.000,C 0.000} C_DIS
LIN {X -32.895,Y -38.771,Z -85.504,A -90.000,B 90.000,C 0.000} C_DIS
LIN {X -32.655,Y -38.767,Z -85.121,A -90.000,B 90.000,C 0.000} C_DIS
LIN {X -32.262,Y -38.755,Z -84.409,A -90.000,B 90.000,C 0.000} C_DIS
LIN {X -31.846,Y -38.744,Z -83.678,A -90.000,B 90.000,C 0.000} C_DIS
LIN {X -31.735,Y -38.735,Z -83.490,A -90.000,B 90.000,C 0.000} C_DIS
LIN {X -31.631,Y -38.727,Z -83.333,A -90.000,B 90.000,C 0.000} C_DIS
LIN {X -31.572,Y -38.722,Z -83.248,A -90.000,B 90.000,C 0.000} C_DIS
LIN {X -31.476,Y -38.717,Z -83.120,A -90.000,B 90.000,C 0.000} C_DIS
LIN {X -31.402,Y -38.714,Z -83.030,A -90.000,B 90.000,C 0.000} C_DIS
LIN {X -31.177,Y -38.705,Z -82.771,A -90.000,B 90.000,C 0.000} C_DIS
LIN {X -31.061,Y -38.701,Z -82.646,A -90.000,B 90.000,C 0.000} C_DIS
LIN {X -30.476,Y -38.681,Z -82.041,A -90.000,B 90.000,C 0.000} C_DIS
LIN {X -30.218,Y -38.674,Z -81.790,A -90.000,B 90.000,C 0.000} C_DIS
LIN {X -29.808,Y -38.635,Z -81.290,A -90.000,B 90.000,C 0.000} C_DIS
LIN {X -29.582,Y -38.612,Z -81.020,A -90.000,B 90.000,C 0.000} C_DIS
LIN {X -29.539,Y -38.607,Z -80.970,A -90.000,B 90.000,C 0.000} C_DIS
LIN {X -29.365,Y -38.592,Z -80.784,A -90.000,B 90.000,C 0.000} C_DIS
LIN {X -29.206,Y -38.578,Z -80.618,A -90.000,B 90.000,C 0.000} C_DIS
LIN {X -29.132,Y -38.572,Z -80.544,A -90.000,B 90.000,C 0.000} C_DIS
LIN {X -28.733,Y -38.544,Z -80.170,A -90.000,B 90.000,C 0.000} C_DIS
LIN {X -28.259,Y -38.497,Z -79.637,A -90.000,B 90.000,C 0.000} C_DIS
LIN {X -27.928,Y -38.443,Z -79.270,A -90.000,B 90.000,C 0.000} C_DIS
LIN {X -27.644,Y -38.392,Z -78.936,A -90.000,B 90.000,C 0.000} C_DIS
LIN {X -27.495,Y -38.366,Z -78.768,A -90.000,B 90.000,C 0.000} C_DIS
LIN {X -27.241,Y -38.325,Z -78.497,A -90.000,B 90.000,C 0.000} C_DIS
LIN {X -26.172,Y -38.160,Z -77.412,A -90.000,B 90.000,C 0.000} C_DIS
LIN {X -25.935,Y -38.121,Z -77.171,A -90.000,B 90.000,C 0.000} C_DIS
LIN {X -25.407,Y -37.996,Z -76.650,A -90.000,B 90.000,C 0.000} C_DIS
LIN {X -24.963,Y -37.895,Z -76.227,A -90.000,B 90.000,C 0.000} C_DIS
LIN {X -24.850,Y -37.871,Z -76.126,A -90.000,B 90.000,C 0.000} C_DIS
LIN {X -24.563,Y -37.815,Z -75.890,A -90.000,B 90.000,C 0.000} C_DIS
LIN {X -23.706,Y -37.672,Z -75.190,A -90.000,B 90.000,C 0.000} C_DIS
LIN {X -23.282,Y -37.585,Z -74.859,A -90.000,B 90.000,C 0.000} C_DIS
LIN {X -23.178,Y -37.561,Z -74.782,A -90.000,B 90.000,C 0.000} C_DIS
LIN {X -22.806,Y -37.511,Z -74.502,A -90.000,B 90.000,C 0.000} C_DIS
LIN {X -22.645,Y -37.492,Z -74.387,A -90.000,B 90.000,C 0.000} C_DIS
LIN {X -22.334,Y -37.483,Z -74.149,A -90.000,B 90.000,C 0.000} C_DIS
LIN {X -22.153,Y -37.480,Z -74.018,A -90.000,B 90.000,C 0.000} C_DIS
LIN {X -21.676,Y -37.478,Z -73.686,A -90.000,B 90.000,C 0.000} C_DIS
LIN {X -21.471,Y -37.486,Z -73.547,A -90.000,B 90.000,C 0.000} C_DIS
LIN {X -21.088,Y -37.510,Z -73.305,A -90.000,B 90.000,C 0.000} C_DIS
LIN {X -20.756,Y -37.534,Z -73.113,A -90.000,B 90.000,C 0.000} C_DIS
LIN {X -20.250,Y -37.535,Z -72.841,A -90.000,B 90.000,C 0.000} C_DIS
LIN {X -20.135,Y -37.533,Z -72.786,A -90.000,B 90.000,C 0.000} C_DIS
LIN {X -19.444,Y -37.527,Z -72.476,A -90.000,B 90.000,C 0.000} C_DIS
LIN {X -18.752,Y -37.537,Z -72.190,A -90.000,B 90.000,C 0.000} C_DIS
LIN {X -18.644,Y -37.539,Z -72.147,A -90.000,B 90.000,C 0.000} C_DIS
LIN {X -18.303,Y -37.537,Z -72.019,A -90.000,B 90.000,C 0.000} C_DIS
LIN {X -18.153,Y -37.533,Z -71.967,A -90.000,B 90.000,C 0.000} C_DIS
LIN {X -17.985,Y -37.530,Z -71.913,A -90.000,B 90.000,C 0.000} C_DIS
LIN {X -17.418,Y -37.514,Z -71.755,A -90.000,B 90.000,C 0.000} C_DIS
LIN {X -16.842,Y -37.495,Z -71.597,A -90.000,B 90.000,C 0.000} C_DIS
LIN {X -16.536,Y -37.476,Z -71.522,A -90.000,B 90.000,C 0.000} C_DIS
LIN {X -16.359,Y -37.467,Z -71.482,A -90.000,B 90.000,C 0.000} C_DIS
LIN {X -15.990,Y -37.450,Z -71.407,A -90.000,B 90.000,C 0.000} C_DIS
LIN {X -15.888,Y -37.446,Z -71.390,A -90.000,B 90.000,C 0.000} C_DIS
LIN {X -15.717,Y -37.442,Z -71.367,A -90.000,B 90.000,C 0.000} C_DIS
LIN {X -15.422,Y -37.432,Z -71.331,A -90.000,B 90.000,C 0.000} C_DIS
LIN {X -15.054,Y -37.420,Z -71.300,A -90.000,B 90.000,C 0.000} C_DIS
LIN {X -14.581,Y -37.411,Z -71.271,A -90.000,B 90.000,C 0.000} C_DIS
LIN {X -14.113,Y -37.410,Z -71.259,A -90.000,B 90.000,C 0.000} C_DIS
LIN {X -12.708,Y -37.403,Z -71.227,A -90.000,B 90.000,C 0.000} C_DIS
LIN {X -11.821,Y -37.381,Z -71.239,A -90.000,B 90.000,C 0.000} C_DIS
LIN {X -11.202,Y -37.364,Z -71.250,A -90.000,B 90.000,C 0.000} C_DIS
LIN {X -11.057,Y -37.361,Z -71.257,A -90.000,B 90.000,C 0.000} C_DIS
LIN {X -10.258,Y -37.355,Z -71.309,A -90.000,B 90.000,C 0.000} C_DIS
LIN {X -8.932,Y -37.356,Z -71.411,A -90.000,B 90.000,C 0.000} C_DIS
LIN {X -7.913,Y -37.330,Z -71.510,A -90.000,B 90.000,C 0.000} C_DIS
LIN {X -7.046,Y -37.320,Z -71.613,A -90.000,B 90.000,C 0.000} C_DIS
LIN {X -6.905,Y -37.320,Z -71.630,A -90.000,B 90.000,C 0.000} C_DIS
LIN {X -6.741,Y -37.322,Z -71.655,A -90.000,B 90.000,C 0.000} C_DIS
LIN {X -5.025,Y -37.366,Z -71.949,A -90.000,B 90.000,C 0.000} C_DIS
LIN {X -4.128,Y -37.365,Z -72.116,A -90.000,B 90.000,C 0.000} C_DIS
LIN {X -2.587,Y -37.369,Z -72.385,A -90.000,B 90.000,C 0.000} C_DIS
LIN {X -2.351,Y -37.371,Z -72.427,A -90.000,B 90.000,C 0.000} C_DIS
LIN {X -1.891,Y -37.383,Z -72.520,A -90.000,B 90.000,C 0.000} C_DIS
LIN {X -0.942,Y -37.414,Z -72.709,A -90.000,B 90.000,C 0.000} C_DIS
LIN {X -0.397,Y -37.431,Z -72.814,A -90.000,B 90.000,C 0.000} C_DIS
LIN {X 0.739,Y -37.442,Z -73.045,A -90.000,B 90.000,C 0.000} C_DIS
LIN {X 1.485,Y -37.461,Z -73.194,A -90.000,B 90.000,C 0.000} C_DIS
LIN {X 1.608,Y -37.465,Z -73.218,A -90.000,B 90.000,C 0.000} C_DIS
LIN {X 1.893,Y -37.482,Z -73.273,A -90.000,B 90.000,C 0.000} C_DIS
LIN {X 2.172,Y -37.497,Z -73.322,A -90.000,B 90.000,C 0.000} C_DIS
LIN {X 2.475,Y -37.518,Z -73.383,A -90.000,B 90.000,C 0.000} C_DIS
LIN {X 2.959,Y -37.556,Z -73.480,A -90.000,B 90.000,C 0.000} C_DIS
LIN {X 4.137,Y -37.650,Z -73.719,A -90.000,B 90.000,C 0.000} C_DIS
LIN {X 4.725,Y -37.719,Z -73.831,A -90.000,B 90.000,C 0.000} C_DIS
LIN {X 5.527,Y -37.812,Z -73.973,A -90.000,B 90.000,C 0.000} C_DIS
LIN {X 5.893,Y -37.860,Z -74.037,A -90.000,B 90.000,C 0.000} C_DIS
LIN {X 6.630,Y -37.979,Z -74.162,A -90.000,B 90.000,C 0.000} C_DIS
LIN {X 7.699,Y -38.161,Z -74.372,A -90.000,B 90.000,C 0.000} C_DIS
LIN {X 8.502,Y -38.299,Z -74.530,A -90.000,B 90.000,C 0.000} C_DIS
LIN {X 9.011,Y -38.383,Z -74.614,A -90.000,B 90.000,C 0.000} C_DIS
LIN {X 9.587,Y -38.477,Z -74.704,A -90.000,B 90.000,C 0.000} C_DIS
LIN {X 10.114,Y -38.561,Z -74.773,A -90.000,B 90.000,C 0.000} C_DIS
LIN {X 10.627,Y -38.637,Z -74.840,A -90.000,B 90.000,C 0.000} C_DIS
LIN {X 10.864,Y -38.672,Z -74.879,A -90.000,B 90.000,C 0.000} C_DIS
LIN {X 11.237,Y -38.675,Z -74.484,A -90.000,B 90.000,C 0.000} C_DIS
LIN {X 11.483,Y -38.666,Z -74.239,A -90.000,B 90.000,C 0.000} C_DIS
LIN {X 11.520,Y -38.664,Z -74.204,A -90.000,B 90.000,C 0.000} C_DIS
LIN {X 11.657,Y -38.656,Z -74.086,A -90.000,B 90.000,C 0.000} C_DIS
LIN {X 11.774,Y -38.650,Z -73.991,A -90.000,B 90.000,C 0.000} C_DIS
LIN {X 11.942,Y -38.644,Z -73.869,A -90.000,B 90.000,C 0.000} C_DIS
LIN {X 12.138,Y -38.637,Z -73.741,A -90.000,B 90.000,C 0.000} C_DIS
LIN {X 12.324,Y -38.621,Z -73.625,A -90.000,B 90.000,C 0.000} C_DIS
LIN {X 12.459,Y -38.600,Z -73.543,A -90.000,B 90.000,C 0.000} C_DIS
LIN {X 12.428,Y -38.496,Z -73.144,A -90.000,B 90.000,C 0.000} C_DIS
LIN {X 12.421,Y -38.467,Z -73.034,A -90.000,B 90.000,C 0.000} C_DIS
LIN {X 12.416,Y -38.436,Z -72.917,A -90.000,B 90.000,C 0.000} C_DIS
LIN {X 12.416,Y -38.386,Z -72.725,A -90.000,B 90.000,C 0.000} C_DIS
LIN {X 12.432,Y -38.291,Z -72.379,A -90.000,B 90.000,C 0.000} C_DIS
LIN {X 12.453,Y -38.213,Z -72.120,A -90.000,B 90.000,C 0.000} C_DIS
LIN {X 12.420,Y -38.114,Z -71.790,A -90.000,B 90.000,C 0.000} C_DIS
LIN {X 12.410,Y -38.050,Z -71.583,A -90.000,B 90.000,C 0.000} C_DIS
LIN {X 12.410,Y -37.986,Z -71.376,A -90.000,B 90.000,C 0.000} C_DIS
LIN {X 12.415,Y -37.932,Z -71.199,A -90.000,B 90.000,C 0.000} C_DIS
LIN {X 12.428,Y -37.879,Z -71.028,A -90.000,B 90.000,C 0.000} C_DIS
LIN {X 12.444,Y -37.824,Z -70.849,A -90.000,B 90.000,C 0.000} C_DIS
LIN {X 12.475,Y -37.755,Z -70.625,A -90.000,B 90.000,C 0.000} C_DIS
LIN {X 12.485,Y -37.737,Z -70.566,A -90.000,B 90.000,C 0.000} C_DIS
LIN {X 12.524,Y -37.682,Z -70.391,A -90.000,B 90.000,C 0.000} C_DIS
LIN {X 12.559,Y -37.634,Z -70.261,A -90.000,B 90.000,C 0.000} C_DIS
LIN {X 12.637,Y -37.536,Z -70.034,A -90.000,B 90.000,C 0.000} C_DIS
LIN {X 12.724,Y -37.443,Z -69.822,A -90.000,B 90.000,C 0.000} C_DIS
LIN {X 12.774,Y -37.394,Z -69.713,A -90.000,B 90.000,C 0.000} C_DIS
LIN {X 12.864,Y -37.319,Z -69.547,A -90.000,B 90.000,C 0.000} C_DIS
LIN {X 12.877,Y -37.308,Z -69.525,A -90.000,B 90.000,C 0.000} C_DIS
LIN {X 12.927,Y -37.276,Z -69.438,A -90.000,B 90.000,C 0.000} C_DIS
LIN {X 13.018,Y -37.201,Z -69.270,A -90.000,B 90.000,C 0.000} C_DIS
LIN {X 13.137,Y -37.095,Z -69.028,A -90.000,B 90.000,C 0.000} C_DIS
LIN {X 13.172,Y -37.086,Z -68.950,A -90.000,B 90.000,C 0.000} C_DIS
LIN {X 13.263,Y -37.120,Z -68.724,A -90.000,B 90.000,C 0.000} C_DIS
LIN {X 13.313,Y -37.134,Z -68.580,A -90.000,B 90.000,C 0.000} C_DIS
LIN {X 13.354,Y -37.139,Z -68.441,A -90.000,B 90.000,C 0.000} C_DIS
LIN {X 13.372,Y -37.138,Z -68.374,A -90.000,B 90.000,C 0.000} C_DIS
LIN {X 13.400,Y -37.131,Z -68.243,A -90.000,B 90.000,C 0.000} C_DIS
LIN {X 13.420,Y -37.116,Z -68.116,A -90.000,B 90.000,C 0.000} C_DIS
LIN {X 13.427,Y -37.105,Z -68.055,A -90.000,B 90.000,C 0.000} C_DIS
LIN {X 13.435,Y -37.077,Z -67.937,A -90.000,B 90.000,C 0.000} C_DIS
LIN {X 13.435,Y -37.041,Z -67.823,A -90.000,B 90.000,C 0.000} C_DIS
LIN {X 13.432,Y -37.020,Z -67.768,A -90.000,B 90.000,C 0.000} C_DIS
LIN {X 13.421,Y -36.974,Z -67.662,A -90.000,B 90.000,C 0.000} C_DIS
LIN {X 13.412,Y -36.950,Z -67.610,A -90.000,B 90.000,C 0.000} C_DIS
LIN {X 13.390,Y -36.899,Z -67.511,A -90.000,B 90.000,C 0.000} C_DIS
LIN {X 13.360,Y -36.843,Z -67.416,A -90.000,B 90.000,C 0.000} C_DIS
LIN {X 13.323,Y -36.785,Z -67.326,A -90.000,B 90.000,C 0.000} C_DIS
LIN {X 13.302,Y -36.754,Z -67.283,A -90.000,B 90.000,C 0.000} C_DIS
LIN {X 13.255,Y -36.690,Z -67.200,A -90.000,B 90.000,C 0.000} C_DIS
LIN {X 13.201,Y -36.623,Z -67.121,A -90.000,B 90.000,C 0.000} C_DIS
LIN {X 13.140,Y -36.553,Z -67.047,A -90.000,B 90.000,C 0.000} C_DIS
LIN {X 13.074,Y -36.479,Z -66.977,A -90.000,B 90.000,C 0.000} C_DIS
LIN {X 13.038,Y -36.447,Z -66.943,A -90.000,B 90.000,C 0.000} C_DIS
LIN {X 12.962,Y -36.384,Z -66.880,A -90.000,B 90.000,C 0.000} C_DIS
LIN {X 12.880,Y -36.318,Z -66.820,A -90.000,B 90.000,C 0.000} C_DIS
LIN {X 12.793,Y -36.250,Z -66.765,A -90.000,B 90.000,C 0.000} C_DIS
LIN {X 12.700,Y -36.181,Z -66.714,A -90.000,B 90.000,C 0.000} C_DIS
LIN {X 12.601,Y -36.112,Z -66.666,A -90.000,B 90.000,C 0.000} C_DIS
LIN {X 12.497,Y -36.039,Z -66.623,A -90.000,B 90.000,C 0.000} C_DIS
LIN {X 12.389,Y -36.022,Z -66.583,A -90.000,B 90.000,C 0.000} C_DIS
LIN {X 12.275,Y -36.009,Z -66.548,A -90.000,B 90.000,C 0.000} C_DIS
LIN {X 12.156,Y -35.997,Z -66.516,A -90.000,B 90.000,C 0.000} C_DIS
LIN {X 12.033,Y -35.987,Z -66.488,A -90.000,B 90.000,C 0.000} C_DIS
LIN {X 11.905,Y -35.979,Z -66.463,A -90.000,B 90.000,C 0.000} C_DIS
LIN {X 11.774,Y -35.976,Z -66.442,A -90.000,B 90.000,C 0.000} C_DIS
LIN {X 11.638,Y -35.975,Z -66.424,A -90.000,B 90.000,C 0.000} C_DIS
LIN {X 11.498,Y -35.976,Z -66.410,A -90.000,B 90.000,C 0.000} C_DIS
LIN {X 11.207,Y -35.984,Z -66.392,A -90.000,B 90.000,C 0.000} C_DIS
LIN {X 10.902,Y -36.000,Z -66.387,A -90.000,B 90.000,C 0.000} C_DIS
LIN {X 10.585,Y -36.020,Z -66.395,A -90.000,B 90.000,C 0.000} C_DIS
LIN {X 10.257,Y -36.038,Z -66.414,A -90.000,B 90.000,C 0.000} C_DIS
LIN {X 10.089,Y -36.049,Z -66.428,A -90.000,B 90.000,C 0.000} C_DIS
LIN {X 9.747,Y -36.075,Z -66.465,A -90.000,B 90.000,C 0.000} C_DIS
LIN {X 9.572,Y -36.090,Z -66.488,A -90.000,B 90.000,C 0.000} C_DIS
LIN {X 9.396,Y -36.111,Z -66.513,A -90.000,B 90.000,C 0.000} C_DIS
LIN {X 9.219,Y -36.136,Z -66.541,A -90.000,B 90.000,C 0.000} C_DIS
LIN {X 9.040,Y -36.155,Z -66.571,A -90.000,B 90.000,C 0.000} C_DIS
LIN {X 8.678,Y -36.186,Z -66.639,A -90.000,B 90.000,C 0.000} C_DIS
LIN {X 8.495,Y -36.203,Z -66.676,A -90.000,B 90.000,C 0.000} C_DIS
LIN {X 8.128,Y -36.240,Z -66.758,A -90.000,B 90.000,C 0.000} C_DIS
LIN {X 7.943,Y -36.260,Z -66.802,A -90.000,B 90.000,C 0.000} C_DIS
LIN {X 7.574,Y -36.304,Z -66.896,A -90.000,B 90.000,C 0.000} C_DIS
LIN {X 7.204,Y -36.352,Z -66.999,A -90.000,B 90.000,C 0.000} C_DIS
LIN {X 7.020,Y -36.374,Z -67.053,A -90.000,B 90.000,C 0.000} C_DIS
LIN {X 6.653,Y -36.410,Z -67.166,A -90.000,B 90.000,C 0.000} C_DIS
LIN {X 6.110,Y -36.452,Z -67.349,A -90.000,B 90.000,C 0.000} C_DIS
LIN {X 5.754,Y -36.481,Z -67.478,A -90.000,B 90.000,C 0.000} C_DIS
LIN {X 5.405,Y -36.514,Z -67.612,A -90.000,B 90.000,C 0.000} C_DIS
LIN {X 5.233,Y -36.531,Z -67.682,A -90.000,B 90.000,C 0.000} C_DIS
LIN {X 4.896,Y -36.567,Z -67.823,A -90.000,B 90.000,C 0.000} C_DIS
LIN {X 4.570,Y -36.603,Z -67.970,A -90.000,B 90.000,C 0.000} C_DIS
LIN {X 4.411,Y -36.619,Z -68.044,A -90.000,B 90.000,C 0.000} C_DIS
LIN {X 4.101,Y -36.644,Z -68.196,A -90.000,B 90.000,C 0.000} C_DIS
LIN {X 3.952,Y -36.655,Z -68.273,A -90.000,B 90.000,C 0.000} C_DIS
LIN {X 3.663,Y -36.676,Z -68.428,A -90.000,B 90.000,C 0.000} C_DIS
LIN {X 3.389,Y -36.699,Z -68.587,A -90.000,B 90.000,C 0.000} C_DIS
LIN {X 3.132,Y -36.724,Z -68.747,A -90.000,B 90.000,C 0.000} C_DIS
LIN {X 3.011,Y -36.737,Z -68.827,A -90.000,B 90.000,C 0.000} C_DIS
LIN {X 2.781,Y -36.757,Z -68.989,A -90.000,B 90.000,C 0.000} C_DIS
LIN {X 2.571,Y -36.768,Z -69.151,A -90.000,B 90.000,C 0.000} C_DIS
LIN {X 2.383,Y -36.778,Z -69.314,A -90.000,B 90.000,C 0.000} C_DIS
LIN {X 2.256,Y -36.787,Z -69.435,A -90.000,B 90.000,C 0.000} C_DIS
LIN {X 2.179,Y -36.794,Z -69.516,A -90.000,B 90.000,C 0.000} C_DIS
LIN {X 2.108,Y -36.801,Z -69.596,A -90.000,B 90.000,C 0.000} C_DIS
LIN {X 2.043,Y -36.808,Z -69.677,A -90.000,B 90.000,C 0.000} C_DIS
LIN {X 1.958,Y -36.820,Z -69.796,A -90.000,B 90.000,C 0.000} C_DIS
LIN {X 1.910,Y -36.828,Z -69.875,A -90.000,B 90.000,C 0.000} C_DIS
LIN {X 1.868,Y -36.836,Z -69.954,A -90.000,B 90.000,C 0.000} C_DIS
LIN {X 1.833,Y -36.842,Z -70.032,A -90.000,B 90.000,C 0.000} C_DIS
LIN {X 1.794,Y -36.852,Z -70.148,A -90.000,B 90.000,C 0.000} C_DIS
LIN {X 1.772,Y -36.860,Z -70.262,A -90.000,B 90.000,C 0.000} C_DIS
LIN {X 1.766,Y -36.871,Z -70.374,A -90.000,B 90.000,C 0.000} C_DIS
LIN {X 1.773,Y -36.879,Z -70.448,A -90.000,B 90.000,C 0.000} C_DIS
LIN {X 1.787,Y -36.889,Z -70.521,A -90.000,B 90.000,C 0.000} C_DIS
LIN {X 1.797,Y -36.894,Z -70.557,A -90.000,B 90.000,C 0.000} C_DIS
LIN {X 1.824,Y -36.905,Z -70.628,A -90.000,B 90.000,C 0.000} C_DIS
LIN {X 1.859,Y -36.918,Z -70.698,A -90.000,B 90.000,C 0.000} C_DIS
LIN {X 1.880,Y -36.924,Z -70.732,A -90.000,B 90.000,C 0.000} C_DIS
LIN {X 1.928,Y -36.938,Z -70.800,A -90.000,B 90.000,C 0.000} C_DIS
LIN {X 2.017,Y -36.962,Z -70.900,A -90.000,B 90.000,C 0.000} C_DIS
LIN {X 2.087,Y -36.978,Z -70.965,A -90.000,B 90.000,C 0.000} C_DIS
LIN {X 2.211,Y -37.006,Z -71.059,A -90.000,B 90.000,C 0.000} C_DIS
LIN {X 2.305,Y -37.026,Z -71.121,A -90.000,B 90.000,C 0.000} C_DIS
LIN {X 2.464,Y -37.058,Z -71.209,A -90.000,B 90.000,C 0.000} C_DIS
LIN {X 2.582,Y -37.081,Z -71.266,A -90.000,B 90.000,C 0.000} C_DIS
LIN {X 2.711,Y -37.105,Z -71.321,A -90.000,B 90.000,C 0.000} C_DIS
LIN {X 2.850,Y -37.130,Z -71.375,A -90.000,B 90.000,C 0.000} C_DIS
LIN {X 3.077,Y -37.171,Z -71.451,A -90.000,B 90.000,C 0.000} C_DIS
LIN {X 3.329,Y -37.214,Z -71.523,A -90.000,B 90.000,C 0.000} C_DIS
LIN {X 3.605,Y -37.262,Z -71.591,A -90.000,B 90.000,C 0.000} C_DIS
LIN {X 3.804,Y -37.295,Z -71.633,A -90.000,B 90.000,C 0.000} C_DIS
LIN {X 3.907,Y -37.308,Z -71.653,A -90.000,B 90.000,C 0.000} C_DIS
LIN {X 4.551,Y -37.415,Z -71.776,A -90.000,B 90.000,C 0.000} C_DIS
LIN {X 5.121,Y -37.511,Z -71.882,A -90.000,B 90.000,C 0.000} C_DIS
LIN {X 5.645,Y -37.602,Z -71.971,A -90.000,B 90.000,C 0.000} C_DIS
LIN {X 6.694,Y -37.774,Z -72.150,A -90.000,B 90.000,C 0.000} C_DIS
LIN {X 7.040,Y -37.827,Z -72.210,A -90.000,B 90.000,C 0.000} C_DIS
LIN {X 8.481,Y -38.054,Z -72.495,A -90.000,B 90.000,C 0.000} C_DIS
LIN {X 8.916,Y -38.111,Z -72.582,A -90.000,B 90.000,C 0.000} C_DIS
LIN {X 9.423,Y -38.174,Z -72.667,A -90.000,B 90.000,C 0.000} C_DIS
LIN {X 9.932,Y -38.239,Z -72.748,A -90.000,B 90.000,C 0.000} C_DIS
LIN {X 10.172,Y -38.269,Z -72.780,A -90.000,B 90.000,C 0.000} C_DIS
LIN {X 10.360,Y -38.257,Z -72.616,A -90.000,B 90.000,C 0.000} C_DIS
LIN {X 10.424,Y -38.253,Z -72.563,A -90.000,B 90.000,C 0.000} C_DIS
LIN {X 10.438,Y -38.199,Z -72.248,A -90.000,B 90.000,C 0.000} C_DIS
LIN {X 10.446,Y -38.182,Z -72.150,A -90.000,B 90.000,C 0.000} C_DIS
LIN {X 10.431,Y -38.151,Z -72.004,A -90.000,B 90.000,C 0.000} C_DIS
LIN {X 10.422,Y -38.121,Z -71.885,A -90.000,B 90.000,C 0.000} C_DIS
LIN {X 10.412,Y -38.067,Z -71.675,A -90.000,B 90.000,C 0.000} C_DIS
LIN {X 10.410,Y -38.042,Z -71.578,A -90.000,B 90.000,C 0.000} C_DIS
LIN {X 10.411,Y -37.977,Z -71.321,A -90.000,B 90.000,C 0.000} C_DIS
LIN {X 10.417,Y -37.927,Z -71.122,A -90.000,B 90.000,C 0.000} C_DIS
LIN {X 10.443,Y -37.839,Z -70.774,A -90.000,B 90.000,C 0.000} C_DIS
LIN {X 10.451,Y -37.812,Z -70.675,A -90.000,B 90.000,C 0.000} C_DIS
LIN {X 10.468,Y -37.772,Z -70.537,A -90.000,B 90.000,C 0.000} C_DIS
LIN {X 10.506,Y -37.695,Z -70.276,A -90.000,B 90.000,C 0.000} C_DIS
LIN {X 10.529,Y -37.658,Z -70.156,A -90.000,B 90.000,C 0.000} C_DIS
LIN {X 10.569,Y -37.602,Z -69.975,A -90.000,B 90.000,C 0.000} C_DIS
LIN {X 10.591,Y -37.575,Z -69.887,A -90.000,B 90.000,C 0.000} C_DIS
LIN {X 10.631,Y -37.516,Z -69.742,A -90.000,B 90.000,C 0.000} C_DIS
LIN {X 10.673,Y -37.463,Z -69.613,A -90.000,B 90.000,C 0.000} C_DIS
LIN {X 10.755,Y -37.367,Z -69.380,A -90.000,B 90.000,C 0.000} C_DIS
LIN {X 10.812,Y -37.308,Z -69.237,A -90.000,B 90.000,C 0.000} C_DIS
LIN {X 10.850,Y -37.273,Z -69.141,A -90.000,B 90.000,C 0.000} C_DIS
LIN {X 10.911,Y -37.199,Z -68.956,A -90.000,B 90.000,C 0.000} C_DIS
LIN {X 10.954,Y -37.133,Z -68.784,A -90.000,B 90.000,C 0.000} C_DIS
LIN {X 10.980,Y -37.072,Z -68.623,A -90.000,B 90.000,C 0.000} C_DIS
LIN {X 10.989,Y -37.016,Z -68.473,A -90.000,B 90.000,C 0.000} C_DIS
LIN {X 10.985,Y -36.977,Z -68.368,A -90.000,B 90.000,C 0.000} C_DIS
LIN {X 10.973,Y -36.939,Z -68.269,A -90.000,B 90.000,C 0.000} C_DIS
LIN {X 10.960,Y -36.914,Z -68.207,A -90.000,B 90.000,C 0.000} C_DIS
LIN {X 10.944,Y -36.889,Z -68.147,A -90.000,B 90.000,C 0.000} C_DIS
LIN {X 10.924,Y -36.865,Z -68.089,A -90.000,B 90.000,C 0.000} C_DIS
LIN {X 10.900,Y -36.841,Z -68.034,A -90.000,B 90.000,C 0.000} C_DIS
LIN {X 10.873,Y -36.818,Z -67.982,A -90.000,B 90.000,C 0.000} C_DIS
LIN {X 10.843,Y -36.796,Z -67.932,A -90.000,B 90.000,C 0.000} C_DIS
LIN {X 10.810,Y -36.774,Z -67.885,A -90.000,B 90.000,C 0.000} C_DIS
LIN {X 10.773,Y -36.754,Z -67.840,A -90.000,B 90.000,C 0.000} C_DIS
LIN {X 10.690,Y -36.716,Z -67.757,A -90.000,B 90.000,C 0.000} C_DIS
LIN {X 10.596,Y -36.682,Z -67.684,A -90.000,B 90.000,C 0.000} C_DIS
LIN {X 10.491,Y -36.653,Z -67.619,A -90.000,B 90.000,C 0.000} C_DIS
LIN {X 10.376,Y -36.629,Z -67.563,A -90.000,B 90.000,C 0.000} C_DIS
LIN {X 10.251,Y -36.610,Z -67.516,A -90.000,B 90.000,C 0.000} C_DIS
LIN {X 10.185,Y -36.603,Z -67.496,A -90.000,B 90.000,C 0.000} C_DIS
LIN {X 10.047,Y -36.592,Z -67.461,A -90.000,B 90.000,C 0.000} C_DIS
LIN {X 9.901,Y -36.585,Z -67.433,A -90.000,B 90.000,C 0.000} C_DIS
LIN {X 9.747,Y -36.583,Z -67.414,A -90.000,B 90.000,C 0.000} C_DIS
LIN {X 9.587,Y -36.585,Z -67.401,A -90.000,B 90.000,C 0.000} C_DIS
LIN {X 9.421,Y -36.586,Z -67.396,A -90.000,B 90.000,C 0.000} C_DIS
LIN {X 9.161,Y -36.586,Z -67.400,A -90.000,B 90.000,C 0.000} C_DIS
LIN {X 8.983,Y -36.589,Z -67.411,A -90.000,B 90.000,C 0.000} C_DIS
LIN {X 8.801,Y -36.596,Z -67.429,A -90.000,B 90.000,C 0.000} C_DIS
LIN {X 8.616,Y -36.604,Z -67.451,A -90.000,B 90.000,C 0.000} C_DIS
LIN {X 8.428,Y -36.614,Z -67.480,A -90.000,B 90.000,C 0.000} C_DIS
LIN {X 8.143,Y -36.630,Z -67.532,A -90.000,B 90.000,C 0.000} C_DIS
LIN {X 7.953,Y -36.641,Z -67.574,A -90.000,B 90.000,C 0.000} C_DIS
LIN {X 7.667,Y -36.657,Z -67.644,A -90.000,B 90.000,C 0.000} C_DIS
LIN {X 7.383,Y -36.673,Z -67.724,A -90.000,B 90.000,C 0.000} C_DIS
LIN {X 7.195,Y -36.685,Z -67.782,A -90.000,B 90.000,C 0.000} C_DIS
LIN {X 6.920,Y -36.704,Z -67.875,A -90.000,B 90.000,C 0.000} C_DIS
LIN {X 6.740,Y -36.718,Z -67.941,A -90.000,B 90.000,C 0.000} C_DIS
LIN {X 6.479,Y -36.742,Z -68.046,A -90.000,B 90.000,C 0.000} C_DIS
LIN {X 6.311,Y -36.759,Z -68.119,A -90.000,B 90.000,C 0.000} C_DIS
LIN {X 6.149,Y -36.778,Z -68.195,A -90.000,B 90.000,C 0.000} C_DIS
LIN {X 5.994,Y -36.797,Z -68.272,A -90.000,B 90.000,C 0.000} C_DIS
LIN {X 5.774,Y -36.828,Z -68.391,A -90.000,B 90.000,C 0.000} C_DIS
LIN {X 5.638,Y -36.848,Z -68.472,A -90.000,B 90.000,C 0.000} C_DIS
LIN {X 5.450,Y -36.872,Z -68.595,A -90.000,B 90.000,C 0.000} C_DIS
LIN {X 5.337,Y -36.885,Z -68.678,A -90.000,B 90.000,C 0.000} C_DIS
LIN {X 5.235,Y -36.899,Z -68.761,A -90.000,B 90.000,C 0.000} C_DIS
LIN {X 5.143,Y -36.913,Z -68.844,A -90.000,B 90.000,C 0.000} C_DIS
LIN {X 5.064,Y -36.928,Z -68.927,A -90.000,B 90.000,C 0.000} C_DIS
LIN {X 5.028,Y -36.936,Z -68.969,A -90.000,B 90.000,C 0.000} C_DIS
LIN {X 4.968,Y -36.953,Z -69.051,A -90.000,B 90.000,C 0.000} C_DIS
LIN {X 4.920,Y -36.971,Z -69.132,A -90.000,B 90.000,C 0.000} C_DIS
LIN {X 4.887,Y -36.990,Z -69.213,A -90.000,B 90.000,C 0.000} C_DIS
LIN {X 4.869,Y -37.010,Z -69.292,A -90.000,B 90.000,C 0.000} C_DIS
LIN {X 4.865,Y -37.020,Z -69.330,A -90.000,B 90.000,C 0.000} C_DIS
LIN {X 4.867,Y -37.036,Z -69.388,A -90.000,B 90.000,C 0.000} C_DIS
LIN {X 4.879,Y -37.052,Z -69.444,A -90.000,B 90.000,C 0.000} C_DIS
LIN {X 4.899,Y -37.069,Z -69.499,A -90.000,B 90.000,C 0.000} C_DIS
LIN {X 4.930,Y -37.087,Z -69.553,A -90.000,B 90.000,C 0.000} C_DIS
LIN {X 4.986,Y -37.111,Z -69.622,A -90.000,B 90.000,C 0.000} C_DIS
LIN {X 5.021,Y -37.123,Z -69.656,A -90.000,B 90.000,C 0.000} C_DIS
LIN {X 5.105,Y -37.147,Z -69.721,A -90.000,B 90.000,C 0.000} C_DIS
LIN {X 5.154,Y -37.159,Z -69.752,A -90.000,B 90.000,C 0.000} C_DIS
LIN {X 5.267,Y -37.184,Z -69.812,A -90.000,B 90.000,C 0.000} C_DIS
LIN {X 5.331,Y -37.197,Z -69.841,A -90.000,B 90.000,C 0.000} C_DIS
LIN {X 5.475,Y -37.224,Z -69.895,A -90.000,B 90.000,C 0.000} C_DIS
LIN {X 5.555,Y -37.238,Z -69.921,A -90.000,B 90.000,C 0.000} C_DIS
LIN {X 5.731,Y -37.266,Z -69.969,A -90.000,B 90.000,C 0.000} C_DIS
LIN {X 5.930,Y -37.295,Z -70.012,A -90.000,B 90.000,C 0.000} C_DIS
LIN {X 6.038,Y -37.308,Z -70.032,A -90.000,B 90.000,C 0.000} C_DIS
LIN {X 7.473,Y -37.502,Z -70.285,A -90.000,B 90.000,C 0.000} C_DIS
LIN {X 7.876,Y -37.559,Z -70.366,A -90.000,B 90.000,C 0.000} C_DIS
LIN {X 8.468,Y -37.632,Z -70.486,A -90.000,B 90.000,C 0.000} C_DIS
LIN {X 8.493,Y -37.581,Z -70.283,A -90.000,B 90.000,C 0.000} C_DIS
LIN {X 8.527,Y -37.522,Z -70.046,A -90.000,B 90.000,C 0.000} C_DIS
LIN {X 8.554,Y -37.481,Z -69.887,A -90.000,B 90.000,C 0.000} C_DIS
LIN {X 8.574,Y -37.453,Z -69.785,A -90.000,B 90.000,C 0.000} C_DIS
LIN {X 8.641,Y -37.373,Z -69.492,A -90.000,B 90.000,C 0.000} C_DIS
LIN {X 8.653,Y -37.358,Z -69.442,A -90.000,B 90.000,C 0.000} C_DIS
LIN {X 8.692,Y -37.308,Z -69.297,A -90.000,B 90.000,C 0.000} C_DIS
LIN {X 8.822,Y -37.153,Z -68.836,A -90.000,B 90.000,C 0.000} C_DIS
LIN {X 8.915,Y -37.052,Z -68.538,A -90.000,B 90.000,C 0.000} C_DIS
LIN {X 9.005,Y -36.964,Z -68.278,A -90.000,B 90.000,C 0.000} C_DIS
LIN {X 9.064,Y -36.910,Z -68.125,A -90.000,B 90.000,C 0.000} C_DIS
LIN {X 9.121,Y -36.860,Z -67.988,A -90.000,B 90.000,C 0.000} C_DIS
LIN {X 9.177,Y -36.812,Z -67.866,A -90.000,B 90.000,C 0.000} C_DIS
LIN {X 9.260,Y -36.744,Z -67.710,A -90.000,B 90.000,C 0.000} C_DIS
LIN {X 9.315,Y -36.703,Z -67.623,A -90.000,B 90.000,C 0.000} C_DIS
LIN {X 9.395,Y -36.649,Z -67.516,A -90.000,B 90.000,C 0.000} C_DIS
LIN {X 9.448,Y -36.620,Z -67.461,A -90.000,B 90.000,C 0.000} C_DIS
LIN {X 9.475,Y -36.608,Z -67.437,A -90.000,B 90.000,C 0.000} C_DIS
LIN {X 9.527,Y -36.586,Z -67.399,A -90.000,B 90.000,C 0.000} C_DIS
LIN {X 9.579,Y -36.570,Z -67.372,A -90.000,B 90.000,C 0.000} C_DIS
LIN {X 9.606,Y -36.563,Z -67.362,A -90.000,B 90.000,C 0.000} C_DIS
LIN {X 9.658,Y -36.553,Z -67.349,A -90.000,B 90.000,C 0.000} C_DIS
LIN {X 9.710,Y -36.549,Z -67.346,A -90.000,B 90.000,C 0.000} C_DIS
LIN {X 9.737,Y -36.548,Z -67.348,A -90.000,B 90.000,C 0.000} C_DIS
LIN {X 9.789,Y -36.550,Z -67.358,A -90.000,B 90.000,C 0.000} C_DIS
LIN {X 9.843,Y -36.557,Z -67.375,A -90.000,B 90.000,C 0.000} C_DIS
LIN {X 9.923,Y -36.574,Z -67.416,A -90.000,B 90.000,C 0.000} C_DIS
LIN {X 10.005,Y -36.599,Z -67.470,A -90.000,B 90.000,C 0.000} C_DIS
LIN {X 10.089,Y -36.631,Z -67.537,A -90.000,B 90.000,C 0.000} C_DIS
LIN {X 10.147,Y -36.656,Z -67.588,A -90.000,B 90.000,C 0.000} C_DIS
LIN {X 10.265,Y -36.709,Z -67.702,A -90.000,B 90.000,C 0.000} C_DIS
LIN {X 10.517,Y -36.823,Z -67.960,A -90.000,B 90.000,C 0.000} C_DIS
LIN {X 10.725,Y -36.904,Z -68.164,A -90.000,B 90.000,C 0.000} C_DIS
LIN {X 10.873,Y -36.952,Z -68.296,A -90.000,B 90.000,C 0.000} C_DIS
LIN {X 10.951,Y -36.974,Z -68.359,A -90.000,B 90.000,C 0.000} C_DIS
LIN {X 11.031,Y -36.995,Z -68.419,A -90.000,B 90.000,C 0.000} C_DIS
LIN {X 11.114,Y -37.014,Z -68.476,A -90.000,B 90.000,C 0.000} C_DIS
LIN {X 11.243,Y -37.040,Z -68.554,A -90.000,B 90.000,C 0.000} C_DIS
LIN {X 11.333,Y -37.055,Z -68.600,A -90.000,B 90.000,C 0.000} C_DIS
LIN {X 11.426,Y -37.068,Z -68.641,A -90.000,B 90.000,C 0.000} C_DIS
LIN {X 11.521,Y -37.078,Z -68.676,A -90.000,B 90.000,C 0.000} C_DIS
LIN {X 11.620,Y -37.084,Z -68.705,A -90.000,B 90.000,C 0.000} C_DIS
LIN {X 11.722,Y -37.086,Z -68.727,A -90.000,B 90.000,C 0.000} C_DIS
LIN {X 11.827,Y -37.084,Z -68.741,A -90.000,B 90.000,C 0.000} C_DIS
LIN {X 11.936,Y -37.077,Z -68.746,A -90.000,B 90.000,C 0.000} C_DIS
LIN {X 12.049,Y -37.066,Z -68.744,A -90.000,B 90.000,C 0.000} C_DIS
LIN {X 12.165,Y -37.052,Z -68.731,A -90.000,B 90.000,C 0.000} C_DIS
LIN {X 12.285,Y -37.034,Z -68.709,A -90.000,B 90.000,C 0.000} C_DIS
LIN {X 12.346,Y -37.023,Z -68.694,A -90.000,B 90.000,C 0.000} C_DIS
LIN {X 12.409,Y -37.028,Z -68.677,A -90.000,B 90.000,C 0.000} C_DIS
LIN {X 12.537,Y -37.057,Z -68.633,A -90.000,B 90.000,C 0.000} C_DIS
LIN {X 12.669,Y -37.085,Z -68.578,A -90.000,B 90.000,C 0.000} C_DIS
LIN {X 12.805,Y -37.113,Z -68.511,A -90.000,B 90.000,C 0.000} C_DIS
LIN {X 12.946,Y -37.140,Z -68.431,A -90.000,B 90.000,C 0.000} C_DIS
LIN {X 13.091,Y -37.166,Z -68.337,A -90.000,B 90.000,C 0.000} C_DIS
LIN {X 13.241,Y -37.191,Z -68.230,A -90.000,B 90.000,C 0.000} C_DIS
LIN {X 13.396,Y -37.215,Z -68.108,A -90.000,B 90.000,C 0.000} C_DIS
LIN {X 13.555,Y -37.238,Z -67.971,A -90.000,B 90.000,C 0.000} C_DIS
LIN {X 13.719,Y -37.260,Z -67.819,A -90.000,B 90.000,C 0.000} C_DIS
LIN {X 13.803,Y -37.270,Z -67.737,A -90.000,B 90.000,C 0.000} C_DIS
LIN {X 13.889,Y -37.281,Z -67.650,A -90.000,B 90.000,C 0.000} C_DIS
LIN {X 13.975,Y -37.296,Z -67.560,A -90.000,B 90.000,C 0.000} C_DIS
LIN {X 14.063,Y -37.308,Z -67.465,A -90.000,B 90.000,C 0.000} C_DIS
LIN {X 14.152,Y -37.308,Z -67.366,A -90.000,B 90.000,C 0.000} C_DIS
LIN {X 14.318,Y -37.325,Z -67.179,A -90.000,B 90.000,C 0.000} C_DIS
LIN {X 14.426,Y -37.337,Z -67.066,A -90.000,B 90.000,C 0.000} C_DIS
LIN {X 14.693,Y -37.368,Z -66.817,A -90.000,B 90.000,C 0.000} C_DIS
LIN {X 14.779,Y -37.371,Z -66.743,A -90.000,B 90.000,C 0.000} C_DIS
LIN {X 14.982,Y -37.384,Z -66.584,A -90.000,B 90.000,C 0.000} C_DIS
LIN {X 15.077,Y -37.383,Z -66.516,A -90.000,B 90.000,C 0.000} C_DIS
LIN {X 15.294,Y -37.390,Z -66.378,A -90.000,B 90.000,C 0.000} C_DIS
LIN {X 15.540,Y -37.382,Z -66.236,A -90.000,B 90.000,C 0.000} C_DIS
LIN {X 15.622,Y -37.380,Z -66.193,A -90.000,B 90.000,C 0.000} C_DIS
LIN {X 15.752,Y -37.371,Z -66.132,A -90.000,B 90.000,C 0.000} C_DIS
LIN {X 15.915,Y -37.365,Z -66.064,A -90.000,B 90.000,C 0.000} C_DIS
LIN {X 15.969,Y -37.363,Z -66.042,A -90.000,B 90.000,C 0.000} C_DIS
LIN {X 16.320,Y -37.331,Z -65.921,A -90.000,B 90.000,C 0.000} C_DIS
LIN {X 16.563,Y -37.316,Z -65.847,A -90.000,B 90.000,C 0.000} C_DIS
LIN {X 16.664,Y -37.312,Z -65.821,A -90.000,B 90.000,C 0.000} C_DIS
LIN {X 16.720,Y -37.308,Z -65.804,A -90.000,B 90.000,C 0.000} C_DIS
LIN {X 17.173,Y -37.263,Z -65.663,A -90.000,B 90.000,C 0.000} C_DIS
LIN {X 17.519,Y -37.202,Z -65.557,A -90.000,B 90.000,C 0.000} C_DIS
LIN {X 17.774,Y -37.131,Z -65.482,A -90.000,B 90.000,C 0.000} C_DIS
LIN {X 17.872,Y -37.093,Z -65.454,A -90.000,B 90.000,C 0.000} C_DIS
LIN {X 17.953,Y -37.054,Z -65.433,A -90.000,B 90.000,C 0.000} C_DIS
LIN {X 18.018,Y -37.014,Z -65.417,A -90.000,B 90.000,C 0.000} C_DIS
LIN {X 18.070,Y -36.991,Z -65.407,A -90.000,B 90.000,C 0.000} C_DIS
LIN {X 18.140,Y -36.975,Z -65.399,A -90.000,B 90.000,C 0.000} C_DIS
LIN {X 18.171,Y -36.974,Z -65.403,A -90.000,B 90.000,C 0.000} C_DIS
LIN {X 18.191,Y -36.980,Z -65.414,A -90.000,B 90.000,C 0.000} C_DIS
LIN {X 18.234,Y -37.013,Z -65.461,A -90.000,B 90.000,C 0.000} C_DIS
LIN {X 18.265,Y -37.024,Z -65.481,A -90.000,B 90.000,C 0.000} C_DIS
LIN {X 18.314,Y -37.032,Z -65.499,A -90.000,B 90.000,C 0.000} C_DIS
LIN {X 18.360,Y -37.034,Z -65.510,A -90.000,B 90.000,C 0.000} C_DIS
LIN {X 18.418,Y -37.032,Z -65.519,A -90.000,B 90.000,C 0.000} C_DIS
LIN {X 18.491,Y -37.027,Z -65.525,A -90.000,B 90.000,C 0.000} C_DIS
LIN {X 18.580,Y -37.015,Z -65.529,A -90.000,B 90.000,C 0.000} C_DIS
LIN {X 18.687,Y -36.996,Z -65.529,A -90.000,B 90.000,C 0.000} C_DIS
LIN {X 18.814,Y -36.966,Z -65.525,A -90.000,B 90.000,C 0.000} C_DIS
LIN {X 18.963,Y -37.019,Z -65.517,A -90.000,B 90.000,C 0.000} C_DIS
LIN {X 19.136,Y -37.103,Z -65.503,A -90.000,B 90.000,C 0.000} C_DIS
LIN {X 19.335,Y -37.205,Z -65.485,A -90.000,B 90.000,C 0.000} C_DIS
LIN {X 19.561,Y -37.308,Z -65.460,A -90.000,B 90.000,C 0.000} C_DIS
LIN {X 19.714,Y -37.382,Z -65.443,A -90.000,B 90.000,C 0.000} C_DIS
LIN {X 19.871,Y -37.449,Z -65.434,A -90.000,B 90.000,C 0.000} C_DIS
LIN {X 19.915,Y -37.469,Z -65.434,A -90.000,B 90.000,C 0.000} C_DIS
LIN {X 20.040,Y -37.475,Z -65.324,A -90.000,B 90.000,C 0.000} C_DIS
LIN {X 20.177,Y -37.471,Z -65.216,A -90.000,B 90.000,C 0.000} C_DIS
LIN {X 20.319,Y -37.470,Z -65.109,A -90.000,B 90.000,C 0.000} C_DIS
LIN {X 20.494,Y -37.457,Z -64.992,A -90.000,B 90.000,C 0.000} C_DIS
LIN {X 20.613,Y -37.452,Z -64.919,A -90.000,B 90.000,C 0.000} C_DIS
LIN {X 20.808,Y -37.431,Z -64.815,A -90.000,B 90.000,C 0.000} C_DIS
LIN {X 20.932,Y -37.419,Z -64.752,A -90.000,B 90.000,C 0.000} C_DIS
LIN {X 21.193,Y -37.383,Z -64.643,A -90.000,B 90.000,C 0.000} C_DIS
LIN {X 21.370,Y -37.363,Z -64.575,A -90.000,B 90.000,C 0.000} C_DIS
LIN {X 21.632,Y -37.321,Z -64.496,A -90.000,B 90.000,C 0.000} C_DIS
LIN {X 21.720,Y -37.308,Z -64.472,A -90.000,B 90.000,C 0.000} C_DIS
LIN {X 21.720,Y -60.000,Z -64.472,A -90.000,B 90.000,C 0.000} C_DIS
LIN {X -37.091,Y -60.000,Z -94.157,A -90.000,B 90.000,C 0.000} C_DIS
LIN {X -37.091,Y -37.308,Z -94.157,A -90.000,B 90.000,C 0.000} C_DIS
LIN {X -37.073,Y -37.339,Z -94.032,A -90.000,B 90.000,C 0.000} C_DIS
LIN {X -37.016,Y -37.412,Z -93.686,A -90.000,B 90.000,C 0.000} C_DIS
LIN {X -36.932,Y -37.511,Z -93.237,A -90.000,B 90.000,C 0.000} C_DIS
LIN {X -36.910,Y -37.535,Z -93.134,A -90.000,B 90.000,C 0.000} C_DIS
LIN {X -36.808,Y -37.637,Z -92.691,A -90.000,B 90.000,C 0.000} C_DIS
LIN {X -36.640,Y -37.795,Z -92.033,A -90.000,B 90.000,C 0.000} C_DIS
LIN {X -36.586,Y -37.839,Z -91.828,A -90.000,B 90.000,C 0.000} C_DIS
LIN {X -36.515,Y -37.901,Z -91.517,A -90.000,B 90.000,C 0.000} C_DIS
LIN {X -36.440,Y -37.955,Z -91.200,A -90.000,B 90.000,C 0.000} C_DIS
LIN {X -36.311,Y -38.040,Z -90.707,A -90.000,B 90.000,C 0.000} C_DIS
LIN {X -36.232,Y -38.089,Z -90.440,A -90.000,B 90.000,C 0.000} C_DIS
LIN {X -36.063,Y -38.198,Z -89.815,A -90.000,B 90.000,C 0.000} C_DIS
LIN {X -35.981,Y -38.247,Z -89.540,A -90.000,B 90.000,C 0.000} C_DIS
LIN {X -35.965,Y -38.263,Z -89.397,A -90.000,B 90.000,C 0.000} C_DIS
LIN {X -35.926,Y -38.279,Z -89.117,A -90.000,B 90.000,C 0.000} C_DIS
LIN {X -35.894,Y -38.291,Z -88.931,A -90.000,B 90.000,C 0.000} C_DIS
LIN {X -35.619,Y -38.385,Z -87.563,A -90.000,B 90.000,C 0.000} C_DIS
LIN {X -35.535,Y -38.413,Z -87.163,A -90.000,B 90.000,C 0.000} C_DIS
LIN {X -35.466,Y -38.428,Z -86.841,A -90.000,B 90.000,C 0.000} C_DIS
LIN {X -35.373,Y -38.428,Z -86.419,A -90.000,B 90.000,C 0.000} C_DIS
LIN {X -35.309,Y -38.428,Z -86.158,A -90.000,B 90.000,C 0.000} C_DIS
LIN {X -35.252,Y -38.430,Z -85.957,A -90.000,B 90.000,C 0.000} C_DIS
LIN {X -35.184,Y -38.433,Z -85.747,A -90.000,B 90.000,C 0.000} C_DIS
LIN {X -35.120,Y -38.437,Z -85.570,A -90.000,B 90.000,C 0.000} C_DIS
LIN {X -35.018,Y -38.444,Z -85.319,A -90.000,B 90.000,C 0.000} C_DIS
LIN {X -34.934,Y -38.450,Z -85.132,A -90.000,B 90.000,C 0.000} C_DIS
LIN {X -34.861,Y -38.457,Z -84.983,A -90.000,B 90.000,C 0.000} C_DIS
LIN {X -34.745,Y -38.467,Z -84.760,A -90.000,B 90.000,C 0.000} C_DIS
LIN {X -34.639,Y -38.467,Z -84.570,A -90.000,B 90.000,C 0.000} C_DIS
LIN {X -34.567,Y -38.466,Z -84.450,A -90.000,B 90.000,C 0.000} C_DIS
LIN {X -34.361,Y -38.465,Z -84.121,A -90.000,B 90.000,C 0.000} C_DIS
LIN {X -33.954,Y -38.457,Z -83.384,A -90.000,B 90.000,C 0.000} C_DIS
LIN {X -33.616,Y -38.452,Z -82.789,A -90.000,B 90.000,C 0.000} C_DIS
LIN {X -33.445,Y -38.437,Z -82.497,A -90.000,B 90.000,C 0.000} C_DIS
LIN {X -33.391,Y -38.433,Z -82.410,A -90.000,B 90.000,C 0.000} C_DIS
LIN {X -33.263,Y -38.425,Z -82.218,A -90.000,B 90.000,C 0.000} C_DIS
LIN {X -33.157,Y -38.419,Z -82.066,A -90.000,B 90.000,C 0.000} C_DIS
LIN {X -33.011,Y -38.413,Z -81.874,A -90.000,B 90.000,C 0.000} C_DIS
LIN {X -32.884,Y -38.409,Z -81.721,A -90.000,B 90.000,C 0.000} C_DIS
LIN {X -32.627,Y -38.403,Z -81.427,A -90.000,B 90.000,C 0.000} C_DIS
LIN {X -32.488,Y -38.402,Z -81.278,A -90.000,B 90.000,C 0.000} C_DIS
LIN {X -32.079,Y -38.399,Z -80.852,A -90.000,B 90.000,C 0.000} C_DIS
LIN {X -31.862,Y -38.394,Z -80.628,A -90.000,B 90.000,C 0.000} C_DIS
LIN {X -31.686,Y -38.386,Z -80.456,A -90.000,B 90.000,C 0.000} C_DIS
LIN {X -31.332,Y -38.358,Z -80.025,A -90.000,B 90.000,C 0.000} C_DIS
LIN {X -31.051,Y -38.335,Z -79.689,A -90.000,B 90.000,C 0.000} C_DIS
LIN {X -30.824,Y -38.319,Z -79.443,A -90.000,B 90.000,C 0.000} C_DIS
LIN {X -30.599,Y -38.304,Z -79.210,A -90.000,B 90.000,C 0.000} C_DIS
LIN {X -30.483,Y -38.298,Z -79.096,A -90.000,B 90.000,C 0.000} C_DIS
LIN {X -30.193,Y -38.282,Z -78.822,A -90.000,B 90.000,C 0.000} C_DIS
LIN {X -30.166,Y -38.279,Z -78.797,A -90.000,B 90.000,C 0.000} C_DIS
LIN {X -29.421,Y -38.171,Z -77.966,A -90.000,B 90.000,C 0.000} C_DIS
LIN {X -29.148,Y -38.128,Z -77.644,A -90.000,B 90.000,C 0.000} C_DIS
LIN {X -28.960,Y -38.101,Z -77.432,A -90.000,B 90.000,C 0.000} C_DIS
LIN {X -28.673,Y -38.062,Z -77.125,A -90.000,B 90.000,C 0.000} C_DIS
LIN {X -28.388,Y -38.027,Z -76.835,A -90.000,B 90.000,C 0.000} C_DIS
LIN {X -28.254,Y -38.011,Z -76.698,A -90.000,B 90.000,C 0.000} C_DIS
LIN {X -27.865,Y -37.938,Z -76.306,A -90.000,B 90.000,C 0.000} C_DIS
LIN {X -27.359,Y -37.821,Z -75.798,A -90.000,B 90.000,C 0.000} C_DIS
LIN {X -26.807,Y -37.697,Z -75.253,A -90.000,B 90.000,C 0.000} C_DIS
LIN {X -26.312,Y -37.589,Z -74.782,A -90.000,B 90.000,C 0.000} C_DIS
LIN {X -26.139,Y -37.554,Z -74.631,A -90.000,B 90.000,C 0.000} C_DIS
LIN {X -25.805,Y -37.490,Z -74.357,A -90.000,B 90.000,C 0.000} C_DIS
LIN {X -25.176,Y -37.308,Z -73.861,A -90.000,B 90.000,C 0.000} C_DIS
LIN {X -25.176,Y -60.000,Z -73.861,A -90.000,B 90.000,C 0.000} C_DIS
LIN {X -38.547,Y -60.000,Z -91.631,A -90.000,B 90.000,C 0.000} C_DIS
LIN {X -38.547,Y -37.308,Z -91.631,A -90.000,B 90.000,C 0.000} C_DIS
LIN {X -38.456,Y -37.392,Z -91.276,A -90.000,B 90.000,C 0.000} C_DIS
LIN {X -38.339,Y -37.510,Z -90.751,A -90.000,B 90.000,C 0.000} C_DIS
LIN {X -38.308,Y -37.532,Z -90.623,A -90.000,B 90.000,C 0.000} C_DIS
LIN {X -38.194,Y -37.606,Z -90.189,A -90.000,B 90.000,C 0.000} C_DIS
LIN {X -38.156,Y -37.630,Z -90.052,A -90.000,B 90.000,C 0.000} C_DIS
LIN {X -38.094,Y -37.668,Z -89.843,A -90.000,B 90.000,C 0.000} C_DIS
LIN {X -37.909,Y -37.784,Z -89.165,A -90.000,B 90.000,C 0.000} C_DIS
LIN {X -37.885,Y -37.799,Z -89.085,A -90.000,B 90.000,C 0.000} C_DIS
LIN {X -37.843,Y -37.843,Z -88.748,A -90.000,B 90.000,C 0.000} C_DIS
LIN {X -37.806,Y -37.874,Z -88.518,A -90.000,B 90.000,C 0.000} C_DIS
LIN {X -37.760,Y -37.911,Z -88.267,A -90.000,B 90.000,C 0.000} C_DIS
LIN {X -37.721,Y -37.926,Z -88.076,A -90.000,B 90.000,C 0.000} C_DIS
LIN {X -37.497,Y -37.996,Z -86.969,A -90.000,B 90.000,C 0.000} C_DIS
LIN {X -37.312,Y -38.051,Z -86.090,A -90.000,B 90.000,C 0.000} C_DIS
LIN {X -37.263,Y -38.058,Z -85.872,A -90.000,B 90.000,C 0.000} C_DIS
LIN {X -37.198,Y -38.058,Z -85.613,A -90.000,B 90.000,C 0.000} C_DIS
LIN {X -37.115,Y -38.060,Z -85.333,A -90.000,B 90.000,C 0.000} C_DIS
LIN {X -37.031,Y -38.064,Z -85.074,A -90.000,B 90.000,C 0.000} C_DIS
LIN {X -36.939,Y -38.070,Z -84.823,A -90.000,B 90.000,C 0.000} C_DIS
LIN {X -36.807,Y -38.080,Z -84.502,A -90.000,B 90.000,C 0.000} C_DIS
LIN {X -36.694,Y -38.090,Z -84.252,A -90.000,B 90.000,C 0.000} C_DIS
LIN {X -36.598,Y -38.099,Z -84.057,A -90.000,B 90.000,C 0.000} C_DIS
LIN {X -36.448,Y -38.111,Z -83.774,A -90.000,B 90.000,C 0.000} C_DIS
LIN {X -36.326,Y -38.111,Z -83.556,A -90.000,B 90.000,C 0.000} C_DIS
LIN {X -36.060,Y -38.113,Z -83.124,A -90.000,B 90.000,C 0.000} C_DIS
LIN {X -35.668,Y -38.112,Z -82.414,A -90.000,B 90.000,C 0.000} C_DIS
LIN {X -35.406,Y -38.113,Z -81.950,A -90.000,B 90.000,C 0.000} C_DIS
LIN {X -35.343,Y -38.113,Z -81.839,A -90.000,B 90.000,C 0.000} C_DIS
LIN {X -35.124,Y -38.099,Z -81.465,A -90.000,B 90.000,C 0.000} C_DIS
LIN {X -35.039,Y -38.094,Z -81.328,A -90.000,B 90.000,C 0.000} C_DIS
LIN {X -34.883,Y -38.088,Z -81.094,A -90.000,B 90.000,C 0.000} C_DIS
LIN {X -34.730,Y -38.083,Z -80.878,A -90.000,B 90.000,C 0.000} C_DIS
LIN {X -34.584,Y -38.081,Z -80.685,A -90.000,B 90.000,C 0.000} C_DIS
LIN {X -34.414,Y -38.080,Z -80.477,A -90.000,B 90.000,C 0.000} C_DIS
LIN {X -34.072,Y -38.083,Z -80.082,A -90.000,B 90.000,C 0.000} C_DIS
LIN {X -33.851,Y -38.085,Z -79.846,A -90.000,B 90.000,C 0.000} C_DIS
LIN {X -33.482,Y -38.080,Z -79.462,A -90.000,B 90.000,C 0.000} C_DIS
LIN {X -33.292,Y -38.077,Z -79.266,A -90.000,B 90.000,C 0.000} C_DIS
LIN {X -33.155,Y -38.075,Z -79.131,A -90.000,B 90.000,C 0.000} C_DIS
LIN {X -32.789,Y -38.058,Z -78.684,A -90.000,B 90.000,C 0.000} C_DIS
LIN {X -32.579,Y -38.047,Z -78.432,A -90.000,B 90.000,C 0.000} C_DIS
LIN {X -32.467,Y -38.041,Z -78.306,A -90.000,B 90.000,C 0.000} C_DIS
LIN {X -32.222,Y -38.026,Z -78.042,A -90.000,B 90.000,C 0.000} C_DIS
LIN {X -31.992,Y -38.010,Z -77.805,A -90.000,B 90.000,C 0.000} C_DIS
LIN {X -31.803,Y -37.998,Z -77.622,A -90.000,B 90.000,C 0.000} C_DIS
LIN {X -31.598,Y -37.985,Z -77.429,A -90.000,B 90.000,C 0.000} C_DIS
LIN {X -31.322,Y -37.960,Z -77.117,A -90.000,B 90.000,C 0.000} C_DIS
LIN {X -30.933,Y -37.914,Z -76.682,A -90.000,B 90.000,C 0.000} C_DIS
LIN {X -30.648,Y -37.877,Z -76.345,A -90.000,B 90.000,C 0.000} C_DIS
LIN {X -30.424,Y -37.850,Z -76.093,A -90.000,B 90.000,C 0.000} C_DIS
LIN {X -30.339,Y -37.840,Z -76.002,A -90.000,B 90.000,C 0.000} C_DIS
LIN {X -30.085,Y -37.802,Z -75.733,A -90.000,B 90.000,C 0.000} C_DIS
LIN {X -29.874,Y -37.769,Z -75.519,A -90.000,B 90.000,C 0.000} C_DIS
LIN {X -29.318,Y -37.661,Z -74.959,A -90.000,B 90.000,C 0.000} C_DIS
LIN {X -28.800,Y -37.556,Z -74.437,A -90.000,B 90.000,C 0.000} C_DIS
LIN {X -28.204,Y -37.437,Z -73.846,A -90.000,B 90.000,C 0.000} C_DIS
LIN {X -27.946,Y -37.388,Z -73.600,A -90.000,B 90.000,C 0.000} C_DIS
LIN {X -27.688,Y -37.308,Z -73.358,A -90.000,B 90.000,C 0.000} C_DIS
LIN {X -27.688,Y -60.000,Z -73.358,A -90.000,B 90.000,C 0.000} C_DIS
LIN {X -39.782,Y -60.000,Z -88.647,A -90.000,B 90.000,C 0.000} C_DIS
LIN {X -39.782,Y -37.308,Z -88.647,A -90.000,B 90.000,C 0.000} C_DIS
LIN {X -39.776,Y -37.312,Z -88.624,A -90.000,B 90.000,C 0.000} C_DIS
LIN {X -39.743,Y -37.343,Z -88.375,A -90.000,B 90.000,C 0.000} C_DIS
LIN {X -39.698,Y -37.380,Z -88.097,A -90.000,B 90.000,C 0.000} C_DIS
LIN {X -39.579,Y -37.468,Z -87.456,A -90.000,B 90.000,C 0.000} C_DIS
LIN {X -39.517,Y -37.504,Z -87.133,A -90.000,B 90.000,C 0.000} C_DIS
LIN {X -39.480,Y -37.522,Z -86.942,A -90.000,B 90.000,C 0.000} C_DIS
LIN {X -39.400,Y -37.544,Z -86.554,A -90.000,B 90.000,C 0.000} C_DIS
LIN {X -39.174,Y -37.607,Z -85.486,A -90.000,B 90.000,C 0.000} C_DIS
LIN {X -39.092,Y -37.629,Z -85.137,A -90.000,B 90.000,C 0.000} C_DIS
LIN {X -39.059,Y -37.638,Z -85.011,A -90.000,B 90.000,C 0.000} C_DIS
LIN {X -38.998,Y -37.649,Z -84.797,A -90.000,B 90.000,C 0.000} C_DIS
LIN {X -38.889,Y -37.653,Z -84.460,A -90.000,B 90.000,C 0.000} C_DIS
LIN {X -38.791,Y -37.660,Z -84.190,A -90.000,B 90.000,C 0.000} C_DIS
LIN {X -38.747,Y -37.663,Z -84.071,A -90.000,B 90.000,C 0.000} C_DIS
LIN {X -38.585,Y -37.676,Z -83.680,A -90.000,B 90.000,C 0.000} C_DIS
LIN {X -38.443,Y -37.691,Z -83.369,A -90.000,B 90.000,C 0.000} C_DIS
LIN {X -38.325,Y -37.704,Z -83.129,A -90.000,B 90.000,C 0.000} C_DIS
LIN {X -38.156,Y -37.721,Z -82.809,A -90.000,B 90.000,C 0.000} C_DIS
LIN {X -38.038,Y -37.723,Z -82.597,A -90.000,B 90.000,C 0.000} C_DIS
LIN {X -37.876,Y -37.727,Z -82.330,A -90.000,B 90.000,C 0.000} C_DIS
LIN {X -37.756,Y -37.731,Z -82.135,A -90.000,B 90.000,C 0.000} C_DIS
LIN {X -37.348,Y -37.736,Z -81.394,A -90.000,B 90.000,C 0.000} C_DIS
LIN {X -37.115,Y -37.741,Z -80.980,A -90.000,B 90.000,C 0.000} C_DIS
LIN {X -37.051,Y -37.742,Z -80.868,A -90.000,B 90.000,C 0.000} C_DIS
LIN {X -36.794,Y -37.732,Z -80.427,A -90.000,B 90.000,C 0.000} C_DIS
LIN {X -36.682,Y -37.729,Z -80.249,A -90.000,B 90.000,C 0.000} C_DIS
LIN {X -36.493,Y -37.727,Z -79.963,A -90.000,B 90.000,C 0.000} C_DIS
LIN {X -36.300,Y -37.727,Z -79.691,A -90.000,B 90.000,C 0.000} C_DIS
LIN {X -36.096,Y -37.727,Z -79.425,A -90.000,B 90.000,C 0.000} C_DIS
LIN {X -35.901,Y -37.729,Z -79.186,A -90.000,B 90.000,C 0.000} C_DIS
LIN {X -35.580,Y -37.731,Z -78.816,A -90.000,B 90.000,C 0.000} C_DIS
LIN {X -35.462,Y -37.732,Z -78.685,A -90.000,B 90.000,C 0.000} C_DIS
LIN {X -35.200,Y -37.733,Z -78.408,A -90.000,B 90.000,C 0.000} C_DIS
LIN {X -34.675,Y -37.738,Z -77.862,A -90.000,B 90.000,C 0.000} C_DIS
LIN {X -34.617,Y -37.738,Z -77.804,A -90.000,B 90.000,C 0.000} C_DIS
LIN {X -34.154,Y -37.721,Z -77.239,A -90.000,B 90.000,C 0.000} C_DIS
LIN {X -34.059,Y -37.715,Z -77.128,A -90.000,B 90.000,C 0.000} C_DIS
LIN {X -33.868,Y -37.706,Z -76.916,A -90.000,B 90.000,C 0.000} C_DIS
LIN {X -33.654,Y -37.696,Z -76.686,A -90.000,B 90.000,C 0.000} C_DIS
LIN {X -33.374,Y -37.684,Z -76.396,A -90.000,B 90.000,C 0.000} C_DIS
LIN {X -33.166,Y -37.672,Z -76.195,A -90.000,B 90.000,C 0.000} C_DIS
LIN {X -33.027,Y -37.664,Z -76.064,A -90.000,B 90.000,C 0.000} C_DIS
LIN {X -32.444,Y -37.617,Z -75.405,A -90.000,B 90.000,C 0.000} C_DIS
LIN {X -32.317,Y -37.605,Z -75.255,A -90.000,B 90.000,C 0.000} C_DIS
LIN {X -32.143,Y -37.583,Z -75.050,A -90.000,B 90.000,C 0.000} C_DIS
LIN {X -32.027,Y -37.568,Z -74.919,A -90.000,B 90.000,C 0.000} C_DIS
LIN {X -31.885,Y -37.544,Z -74.761,A -90.000,B 90.000,C 0.000} C_DIS
LIN {X -31.515,Y -37.486,Z -74.371,A -90.000,B 90.000,C 0.000} C_DIS
LIN {X -30.711,Y -37.363,Z -73.555,A -90.000,B 90.000,C 0.000} C_DIS
LIN {X -30.412,Y -37.308,Z -73.252,A -90.000,B 90.000,C 0.000} C_DIS
LIN {X -30.412,Y -60.000,Z -73.252,A -90.000,B 90.000,C 0.000} C_DIS
LIN {X -39.532,Y -60.000,Z -81.290,A -90.000,B 90.000,C 0.000} C_DIS
LIN {X -39.532,Y -37.308,Z -81.290,A -90.000,B 90.000,C 0.000} C_DIS
LIN {X -39.450,Y -37.313,Z -81.155,A -90.000,B 90.000,C 0.000} C_DIS
LIN {X -39.040,Y -37.329,Z -80.407,A -90.000,B 90.000,C 0.000} C_DIS
LIN {X -38.818,Y -37.334,Z -80.015,A -90.000,B 90.000,C 0.000} C_DIS
LIN {X -38.724,Y -37.333,Z -79.849,A -90.000,B 90.000,C 0.000} C_DIS
LIN {X -38.430,Y -37.327,Z -79.349,A -90.000,B 90.000,C 0.000} C_DIS
LIN {X -38.343,Y -37.326,Z -79.210,A -90.000,B 90.000,C 0.000} C_DIS
LIN {X -38.127,Y -37.326,Z -78.882,A -90.000,B 90.000,C 0.000} C_DIS
LIN {X -37.900,Y -37.329,Z -78.559,A -90.000,B 90.000,C 0.000} C_DIS
LIN {X -37.621,Y -37.335,Z -78.191,A -90.000,B 90.000,C 0.000} C_DIS
LIN {X -37.382,Y -37.340,Z -77.900,A -90.000,B 90.000,C 0.000} C_DIS
LIN {X -37.034,Y -37.350,Z -77.497,A -90.000,B 90.000,C 0.000} C_DIS
LIN {X -36.847,Y -37.356,Z -77.291,A -90.000,B 90.000,C 0.000} C_DIS
LIN {X -36.607,Y -37.360,Z -77.037,A -90.000,B 90.000,C 0.000} C_DIS
LIN {X -36.075,Y -37.369,Z -76.482,A -90.000,B 90.000,C 0.000} C_DIS
LIN {X -35.886,Y -37.366,Z -76.250,A -90.000,B 90.000,C 0.000} C_DIS
LIN {X -35.576,Y -37.357,Z -75.874,A -90.000,B 90.000,C 0.000} C_DIS
LIN {X -35.336,Y -37.347,Z -75.606,A -90.000,B 90.000,C 0.000} C_DIS
LIN {X -35.105,Y -37.339,Z -75.356,A -90.000,B 90.000,C 0.000} C_DIS
LIN {X -34.753,Y -37.329,Z -74.991,A -90.000,B 90.000,C 0.000} C_DIS
LIN {X -34.455,Y -37.323,Z -74.703,A -90.000,B 90.000,C 0.000} C_DIS
LIN {X -34.224,Y -37.310,Z -74.441,A -90.000,B 90.000,C 0.000} C_DIS
LIN {X -34.204,Y -37.308,Z -74.418,A -90.000,B 90.000,C 0.000} C_DIS
LIN {X -34.204,Y -60.000,Z -74.418,A -90.000,B 90.000,C 0.000} C_DIS
LIN {X -87.660,Y -60.000,Z -243.561,A -90.000,B 90.000,C 0.000} C_DIS
LIN {X -87.660,Y -37.845,Z -243.561,A -90.000,B 90.000,C 0.000} C_DIS
LIN {X -87.642,Y -37.805,Z -243.485,A -90.000,B 90.000,C 0.000} C_DIS
LIN {X -87.603,Y -37.741,Z -243.355,A -90.000,B 90.000,C 0.000} C_DIS
LIN {X -87.422,Y -37.500,Z -242.849,A -90.000,B 90.000,C 0.000} C_DIS
LIN {X -87.355,Y -37.426,Z -242.684,A -90.000,B 90.000,C 0.000} C_DIS
LIN {X -87.282,Y -37.367,Z -242.543,A -90.000,B 90.000,C 0.000} C_DIS
LIN {X -87.198,Y -37.308,Z -242.392,A -90.000,B 90.000,C 0.000} C_DIS
LIN {X -87.124,Y -37.250,Z -242.245,A -90.000,B 90.000,C 0.000} C_DIS
LIN {X -87.097,Y -37.223,Z -242.185,A -90.000,B 90.000,C 0.000} C_DIS
LIN {X -87.078,Y -37.199,Z -242.132,A -90.000,B 90.000,C 0.000} C_DIS
LIN {X -87.065,Y -37.176,Z -242.087,A -90.000,B 90.000,C 0.000} C_DIS
LIN {X -87.059,Y -37.155,Z -242.049,A -90.000,B 90.000,C 0.000} C_DIS
LIN {X -87.062,Y -37.126,Z -242.005,A -90.000,B 90.000,C 0.000} C_DIS
LIN {X -87.079,Y -37.101,Z -241.975,A -90.000,B 90.000,C 0.000} C_DIS
LIN {X -87.109,Y -37.078,Z -241.958,A -90.000,B 90.000,C 0.000} C_DIS
LIN {X -87.134,Y -37.066,Z -241.955,A -90.000,B 90.000,C 0.000} C_DIS
LIN {X -87.164,Y -37.055,Z -241.958,A -90.000,B 90.000,C 0.000} C_DIS
LIN {X -87.218,Y -37.041,Z -241.971,A -90.000,B 90.000,C 0.000} C_DIS
LIN {X -87.260,Y -37.033,Z -241.985,A -90.000,B 90.000,C 0.000} C_DIS
LIN {X -87.355,Y -37.022,Z -242.030,A -90.000,B 90.000,C 0.000} C_DIS
LIN {X -87.464,Y -37.016,Z -242.093,A -90.000,B 90.000,C 0.000} C_DIS
LIN {X -87.584,Y -37.013,Z -242.169,A -90.000,B 90.000,C 0.000} C_DIS
LIN {X -87.714,Y -37.013,Z -242.259,A -90.000,B 90.000,C 0.000} C_DIS
LIN {X -87.921,Y -37.021,Z -242.413,A -90.000,B 90.000,C 0.000} C_DIS
LIN {X -88.065,Y -37.031,Z -242.526,A -90.000,B 90.000,C 0.000} C_DIS
LIN {X -88.356,Y -37.059,Z -242.768,A -90.000,B 90.000,C 0.000} C_DIS
LIN {X -88.500,Y -37.075,Z -242.891,A -90.000,B 90.000,C 0.000} C_DIS
LIN {X -88.639,Y -37.093,Z -243.014,A -90.000,B 90.000,C 0.000} C_DIS
LIN {X -88.896,Y -37.133,Z -243.251,A -90.000,B 90.000,C 0.000} C_DIS
LIN {X -89.110,Y -37.175,Z -243.463,A -90.000,B 90.000,C 0.000} C_DIS
LIN {X -89.196,Y -37.195,Z -243.553,A -90.000,B 90.000,C 0.000} C_DIS
LIN {X -89.291,Y -37.225,Z -243.665,A -90.000,B 90.000,C 0.000} C_DIS
LIN {X -89.329,Y -37.244,Z -243.720,A -90.000,B 90.000,C 0.000} C_DIS
LIN {X -89.340,Y -37.252,Z -243.741,A -90.000,B 90.000,C 0.000} C_DIS
LIN {X -89.345,Y -37.261,Z -243.757,A -90.000,B 90.000,C 0.000} C_DIS
LIN {X -89.344,Y -37.268,Z -243.769,A -90.000,B 90.000,C 0.000} C_DIS
LIN {X -89.337,Y -37.276,Z -243.775,A -90.000,B 90.000,C 0.000} C_DIS
LIN {X -89.330,Y -37.279,Z -243.776,A -90.000,B 90.000,C 0.000} C_DIS
LIN {X -89.302,Y -37.289,Z -243.771,A -90.000,B 90.000,C 0.000} C_DIS
LIN {X -89.274,Y -37.294,Z -243.761,A -90.000,B 90.000,C 0.000} C_DIS
LIN {X -89.196,Y -37.303,Z -243.721,A -90.000,B 90.000,C 0.000} C_DIS
LIN {X -89.086,Y -37.308,Z -243.654,A -90.000,B 90.000,C 0.000} C_DIS
LIN {X -88.939,Y -37.308,Z -243.561,A -90.000,B 90.000,C 0.000} C_DIS
LIN {X -87.960,Y -37.308,Z -242.895,A -90.000,B 90.000,C 0.000} C_DIS
LIN {X -85.068,Y -37.308,Z -240.988,A -90.000,B 90.000,C 0.000} C_DIS
LIN {X -81.571,Y -37.308,Z -238.798,A -90.000,B 90.000,C 0.000} C_DIS
LIN {X -76.915,Y -37.308,Z -235.965,A -90.000,B 90.000,C 0.000} C_DIS
LIN {X -75.282,Y -37.308,Z -235.028,A -90.000,B 90.000,C 0.000} C_DIS
LIN {X -70.869,Y -37.308,Z -232.540,A -90.000,B 90.000,C 0.000} C_DIS
LIN {X -69.001,Y -37.308,Z -231.500,A -90.000,B 90.000,C 0.000} C_DIS
LIN {X -68.583,Y -37.308,Z -231.271,A -90.000,B 90.000,C 0.000} C_DIS
LIN {X -68.395,Y -37.308,Z -231.170,A -90.000,B 90.000,C 0.000} C_DIS
LIN {X -59.595,Y -37.308,Z -226.639,A -90.000,B 90.000,C 0.000} C_DIS
LIN {X -52.430,Y -37.308,Z -223.071,A -90.000,B 90.000,C 0.000} C_DIS
LIN {X -49.127,Y -37.308,Z -221.440,A -90.000,B 90.000,C 0.000} C_DIS
LIN {X -43.469,Y -37.308,Z -218.670,A -90.000,B 90.000,C 0.000} C_DIS
LIN {X -41.282,Y -37.308,Z -217.574,A -90.000,B 90.000,C 0.000} C_DIS
LIN {X -39.343,Y -37.308,Z -216.606,A -90.000,B 90.000,C 0.000} C_DIS
LIN {X -36.349,Y -37.308,Z -215.120,A -90.000,B 90.000,C 0.000} C_DIS
LIN {X -35.277,Y -37.308,Z -214.565,A -90.000,B 90.000,C 0.000} C_DIS
LIN {X -31.754,Y -37.308,Z -212.699,A -90.000,B 90.000,C 0.000} C_DIS
LIN {X -30.826,Y -37.308,Z -212.213,A -90.000,B 90.000,C 0.000} C_DIS
LIN {X -28.933,Y -37.308,Z -211.157,A -90.000,B 90.000,C 0.000} C_DIS
LIN {X -26.733,Y -37.308,Z -209.956,A -90.000,B 90.000,C 0.000} C_DIS
LIN {X -26.028,Y -37.308,Z -209.562,A -90.000,B 90.000,C 0.000} C_DIS
LIN {X -23.237,Y -37.308,Z -207.905,A -90.000,B 90.000,C 0.000} C_DIS
LIN {X -21.674,Y -37.308,Z -206.953,A -90.000,B 90.000,C 0.000} C_DIS
LIN {X -19.919,Y -37.308,Z -205.807,A -90.000,B 90.000,C 0.000} C_DIS
LIN {X -17.754,Y -37.308,Z -204.362,A -90.000,B 90.000,C 0.000} C_DIS
LIN {X -14.766,Y -37.308,Z -202.201,A -90.000,B 90.000,C 0.000} C_DIS
LIN {X -14.248,Y -37.308,Z -201.828,A -90.000,B 90.000,C 0.000} C_DIS
LIN {X -10.736,Y -37.308,Z -199.100,A -90.000,B 90.000,C 0.000} C_DIS
LIN {X -8.789,Y -37.308,Z -197.501,A -90.000,B 90.000,C 0.000} C_DIS
LIN {X -7.176,Y -37.308,Z -196.190,A -90.000,B 90.000,C 0.000} C_DIS
LIN {X -6.970,Y -37.308,Z -196.013,A -90.000,B 90.000,C 0.000} C_DIS
LIN {X -3.530,Y -37.308,Z -193.099,A -90.000,B 90.000,C 0.000} C_DIS
LIN {X -0.646,Y -37.308,Z -190.606,A -90.000,B 90.000,C 0.000} C_DIS
LIN {X 0.231,Y -37.308,Z -189.813,A -90.000,B 90.000,C 0.000} C_DIS
LIN {X 2.716,Y -37.308,Z -187.615,A -90.000,B 90.000,C 0.000} C_DIS
LIN {X 3.943,Y -37.308,Z -186.468,A -90.000,B 90.000,C 0.000} C_DIS
LIN {X 5.999,Y -37.308,Z -184.607,A -90.000,B 90.000,C 0.000} C_DIS
LIN {X 7.454,Y -37.308,Z -183.224,A -90.000,B 90.000,C 0.000} C_DIS
LIN {X 9.115,Y -37.308,Z -181.685,A -90.000,B 90.000,C 0.000} C_DIS
LIN {X 10.629,Y -37.308,Z -180.240,A -90.000,B 90.000,C 0.000} C_DIS
LIN {X 12.035,Y -37.308,Z -178.914,A -90.000,B 90.000,C 0.000} C_DIS
LIN {X 13.339,Y -37.308,Z -177.677,A -90.000,B 90.000,C 0.000} C_DIS
LIN {X 14.520,Y -37.308,Z -176.552,A -90.000,B 90.000,C 0.000} C_DIS
LIN {X 16.460,Y -37.308,Z -174.629,A -90.000,B 90.000,C 0.000} C_DIS
LIN {X 17.667,Y -37.308,Z -173.339,A -90.000,B 90.000,C 0.000} C_DIS
LIN {X 18.175,Y -37.308,Z -172.793,A -90.000,B 90.000,C 0.000} C_DIS
LIN {X 19.013,Y -37.308,Z -171.793,A -90.000,B 90.000,C 0.000} C_DIS
LIN {X 19.254,Y -37.308,Z -171.501,A -90.000,B 90.000,C 0.000} C_DIS
LIN {X 20.571,Y -37.308,Z -169.691,A -90.000,B 90.000,C 0.000} C_DIS
LIN {X 21.459,Y -37.308,Z -168.313,A -90.000,B 90.000,C 0.000} C_DIS
LIN {X 21.733,Y -37.308,Z -167.735,A -90.000,B 90.000,C 0.000} C_DIS
LIN {X 22.208,Y -37.308,Z -166.906,A -90.000,B 90.000,C 0.000} C_DIS
LIN {X 22.477,Y -37.308,Z -166.189,A -90.000,B 90.000,C 0.000} C_DIS
LIN {X 22.636,Y -37.308,Z -165.470,A -90.000,B 90.000,C 0.000} C_DIS
LIN {X 22.638,Y -37.308,Z -165.460,A -90.000,B 90.000,C 0.000} C_DIS
LIN {X 22.696,Y -37.308,Z -164.543,A -90.000,B 90.000,C 0.000} C_DIS
LIN {X 22.660,Y -37.308,Z -164.493,A -90.000,B 90.000,C 0.000} C_DIS
LIN {X 22.399,Y -37.308,Z -164.028,A -90.000,B 90.000,C 0.000} C_DIS
LIN {X 22.321,Y -37.308,Z -163.805,A -90.000,B 90.000,C 0.000} C_DIS
LIN {X 22.182,Y -37.308,Z -163.291,A -90.000,B 90.000,C 0.000} C_DIS
LIN {X 21.755,Y -37.308,Z -162.870,A -90.000,B 90.000,C 0.000} C_DIS
LIN {X 21.609,Y -37.308,Z -162.716,A -90.000,B 90.000,C 0.000} C_DIS
LIN {X 21.485,Y -37.308,Z -162.513,A -90.000,B 90.000,C 0.000} C_DIS
LIN {X 21.321,Y -37.308,Z -162.161,A -90.000,B 90.000,C 0.000} C_DIS
LIN {X 20.664,Y -37.308,Z -161.371,A -90.000,B 90.000,C 0.000} C_DIS
LIN {X 20.408,Y -37.308,Z -161.007,A -90.000,B 90.000,C 0.000} C_DIS
LIN {X 20.276,Y -37.308,Z -160.759,A -90.000,B 90.000,C 0.000} C_DIS
LIN {X 20.232,Y -37.308,Z -160.668,A -90.000,B 90.000,C 0.000} C_DIS
LIN {X 20.215,Y -37.308,Z -160.617,A -90.000,B 90.000,C 0.000} C_DIS
LIN {X 20.088,Y -37.308,Z -160.387,A -90.000,B 90.000,C 0.000} C_DIS
LIN {X 19.955,Y -37.308,Z -160.138,A -90.000,B 90.000,C 0.000} C_DIS
LIN {X 19.568,Y -37.308,Z -159.330,A -90.000,B 90.000,C 0.000} C_DIS
LIN {X 19.511,Y -37.308,Z -159.173,A -90.000,B 90.000,C 0.000} C_DIS
LIN {X 19.433,Y -37.308,Z -158.932,A -90.000,B 90.000,C 0.000} C_DIS
LIN {X 19.082,Y -37.308,Z -157.676,A -90.000,B 90.000,C 0.000} C_DIS
LIN {X 18.932,Y -37.308,Z -157.213,A -90.000,B 90.000,C 0.000} C_DIS
LIN {X 18.754,Y -37.308,Z -156.274,A -90.000,B 90.000,C 0.000} C_DIS
LIN {X 18.715,Y -37.308,Z -155.995,A -90.000,B 90.000,C 0.000} C_DIS
LIN {X 18.607,Y -37.308,Z -155.043,A -90.000,B 90.000,C 0.000} C_DIS
LIN {X 18.551,Y -37.308,Z -154.591,A -90.000,B 90.000,C 0.000} C_DIS
LIN {X 18.565,Y -37.308,Z -154.282,A -90.000,B 90.000,C 0.000} C_DIS
LIN {X 18.635,Y -37.308,Z -153.377,A -90.000,B 90.000,C 0.000} C_DIS
LIN {X 18.725,Y -37.308,Z -152.878,A -90.000,B 90.000,C 0.000} C_DIS
LIN {X 18.786,Y -37.308,Z -152.602,A -90.000,B 90.000,C 0.000} C_DIS
LIN {X 18.898,Y -37.308,Z -152.300,A -90.000,B 90.000,C 0.000} C_DIS
LIN {X 19.007,Y -37.308,Z -152.040,A -90.000,B 90.000,C 0.000} C_DIS
LIN {X 19.411,Y -37.308,Z -151.218,A -90.000,B 90.000,C 0.000} C_DIS
LIN {X 20.158,Y -37.308,Z -149.734,A -90.000,B 90.000,C 0.000} C_DIS
LIN {X 20.248,Y -37.308,Z -149.576,A -90.000,B 90.000,C 0.000} C_DIS
LIN {X 20.400,Y -37.308,Z -149.339,A -90.000,B 90.000,C 0.000} C_DIS
LIN {X 20.800,Y -37.308,Z -148.833,A -90.000,B 90.000,C 0.000} C_DIS
LIN {X 21.241,Y -37.308,Z -148.288,A -90.000,B 90.000,C 0.000} C_DIS
LIN {X 20.343,Y -37.308,Z -148.653,A -90.000,B 90.000,C 0.000} C_DIS
LIN {X 18.118,Y -37.308,Z -149.496,A -90.000,B 90.000,C 0.000} C_DIS
LIN {X 17.607,Y -37.308,Z -149.673,A -90.000,B 90.000,C 0.000} C_DIS
LIN {X 15.422,Y -37.308,Z -150.392,A -90.000,B 90.000,C 0.000} C_DIS
LIN {X 14.356,Y -37.308,Z -150.729,A -90.000,B 90.000,C 0.000} C_DIS
LIN {X 13.536,Y -37.308,Z -150.959,A -90.000,B 90.000,C 0.000} C_DIS
LIN {X 12.818,Y -37.308,Z -151.149,A -90.000,B 90.000,C 0.000} C_DIS
LIN {X 11.297,Y -37.308,Z -151.524,A -90.000,B 90.000,C 0.000} C_DIS
LIN {X 10.584,Y -37.308,Z -151.694,A -90.000,B 90.000,C 0.000} C_DIS
LIN {X 10.146,Y -37.308,Z -151.791,A -90.000,B 90.000,C 0.000} C_DIS
LIN {X 9.903,Y -37.308,Z -151.828,A -90.000,B 90.000,C 0.000} C_DIS
LIN {X 7.499,Y -37.308,Z -152.207,A -90.000,B 90.000,C 0.000} C_DIS
LIN {X 7.061,Y -37.308,Z -152.254,A -90.000,B 90.000,C 0.000} C_DIS
LIN {X 6.166,Y -37.308,Z -152.299,A -90.000,B 90.000,C 0.000} C_DIS
LIN {X 4.107,Y -37.308,Z -152.427,A -90.000,B 90.000,C 0.000} C_DIS
LIN {X 3.666,Y -37.308,Z -152.424,A -90.000,B 90.000,C 0.000} C_DIS
LIN {X 2.201,Y -37.308,Z -152.336,A -90.000,B 90.000,C 0.000} C_DIS
LIN {X 0.492,Y -37.308,Z -152.256,A -90.000,B 90.000,C 0.000} C_DIS
LIN {X 0.055,Y -37.308,Z -152.203,A -90.000,B 90.000,C 0.000} C_DIS
LIN {X -1.917,Y -37.308,Z -151.848,A -90.000,B 90.000,C 0.000} C_DIS
LIN {X -3.298,Y -37.308,Z -151.610,A -90.000,B 90.000,C 0.000} C_DIS
LIN {X -3.459,Y -37.308,Z -151.576,A -90.000,B 90.000,C 0.000} C_DIS
LIN {X -3.726,Y -37.308,Z -151.508,A -90.000,B 90.000,C 0.000} C_DIS
LIN {X -5.626,Y -37.308,Z -150.950,A -90.000,B 90.000,C 0.000} C_DIS
LIN {X -7.407,Y -37.308,Z -150.431,A -90.000,B 90.000,C 0.000} C_DIS
LIN {X -7.831,Y -37.308,Z -150.263,A -90.000,B 90.000,C 0.000} C_DIS
LIN {X -11.427,Y -37.308,Z -148.795,A -90.000,B 90.000,C 0.000} C_DIS
LIN {X -14.013,Y -37.308,Z -147.428,A -90.000,B 90.000,C 0.000} C_DIS
LIN {X -15.400,Y -37.308,Z -146.690,A -90.000,B 90.000,C 0.000} C_DIS
LIN {X -15.507,Y -37.308,Z -146.621,A -90.000,B 90.000,C 0.000} C_DIS
LIN {X -18.493,Y -37.308,Z -144.619,A -90.000,B 90.000,C 0.000} C_DIS
LIN {X -19.221,Y -37.308,Z -144.134,A -90.000,B 90.000,C 0.000} C_DIS
LIN {X -19.411,Y -37.308,Z -144.004,A -90.000,B 90.000,C 0.000} C_DIS
LIN {X -20.170,Y -37.308,Z -143.396,A -90.000,B 90.000,C 0.000} C_DIS
LIN {X -21.350,Y -37.308,Z -142.462,A -90.000,B 90.000,C 0.000} C_DIS
LIN {X -22.673,Y -37.308,Z -141.395,A -90.000,B 90.000,C 0.000} C_DIS
LIN {X -22.890,Y -37.308,Z -141.217,A -90.000,B 90.000,C 0.000} C_DIS
LIN {X -23.015,Y -37.308,Z -141.110,A -90.000,B 90.000,C 0.000} C_DIS
LIN {X -23.658,Y -37.308,Z -140.492,A -90.000,B 90.000,C 0.000} C_DIS
LIN {X -25.896,Y -37.308,Z -138.240,A -90.000,B 90.000,C 0.000} C_DIS
LIN {X -26.203,Y -37.308,Z -137.924,A -90.000,B 90.000,C 0.000} C_DIS
LIN {X -28.289,Y -37.308,Z -135.409,A -90.000,B 90.000,C 0.000} C_DIS
LIN {X -28.696,Y -37.308,Z -134.912,A -90.000,B 90.000,C 0.000} C_DIS
LIN {X -28.900,Y -37.308,Z -134.647,A -90.000,B 90.000,C 0.000} C_DIS
LIN {X -29.970,Y -37.308,Z -133.041,A -90.000,B 90.000,C 0.000} C_DIS
LIN {X -30.201,Y -37.308,Z -132.686,A -90.000,B 90.000,C 0.000} C_DIS
LIN {X -30.930,Y -37.308,Z -131.535,A -90.000,B 90.000,C 0.000} C_DIS
LIN {X -31.053,Y -37.308,Z -131.320,A -90.000,B 90.000,C 0.000} C_DIS
LIN {X -31.638,Y -37.308,Z -130.198,A -90.000,B 90.000,C 0.000} C_DIS
LIN {X -32.611,Y -37.308,Z -128.296,A -90.000,B 90.000,C 0.000} C_DIS
LIN {X -32.990,Y -37.308,Z -127.443,A -90.000,B 90.000,C 0.000} C_DIS
LIN {X -33.834,Y -37.308,Z -125.482,A -90.000,B 90.000,C 0.000} C_DIS
LIN {X -33.949,Y -37.308,Z -125.205,A -90.000,B 90.000,C 0.000} C_DIS
LIN {X -34.370,Y -37.308,Z -124.048,A -90.000,B 90.000,C 0.000} C_DIS
LIN {X -34.848,Y -37.308,Z -122.723,A -90.000,B 90.000,C 0.000} C_DIS
LIN {X -35.086,Y -37.308,Z -121.891,A -90.000,B 90.000,C 0.000} C_DIS
LIN {X -35.628,Y -37.308,Z -120.186,A -90.000,B 90.000,C 0.000} C_DIS
LIN {X -35.736,Y -37.308,Z -119.797,A -90.000,B 90.000,C 0.000} C_DIS
LIN {X -35.778,Y -37.308,Z -119.602,A -90.000,B 90.000,C 0.000} C_DIS
LIN {X -35.962,Y -37.308,Z -118.933,A -90.000,B 90.000,C 0.000} C_DIS
LIN {X -36.366,Y -37.308,Z -117.169,A -90.000,B 90.000,C 0.000} C_DIS
LIN {X -36.564,Y -37.308,Z -115.782,A -90.000,B 90.000,C 0.000} C_DIS
LIN {X -36.898,Y -37.308,Z -114.044,A -90.000,B 90.000,C 0.000} C_DIS
LIN {X -36.954,Y -37.308,Z -113.666,A -90.000,B 90.000,C 0.000} C_DIS
LIN {X -36.960,Y -37.308,Z -113.586,A -90.000,B 90.000,C 0.000} C_DIS
LIN {X -36.980,Y -37.308,Z -113.428,A -90.000,B 90.000,C 0.000} C_DIS
LIN {X -37.097,Y -37.308,Z -111.879,A -90.000,B 90.000,C 0.000} C_DIS
LIN {X -37.121,Y -37.308,Z -111.317,A -90.000,B 90.000,C 0.000} C_DIS
LIN {X -37.148,Y -37.308,Z -110.942,A -90.000,B 90.000,C 0.000} C_DIS
LIN {X -37.140,Y -37.308,Z -110.405,A -90.000,B 90.000,C 0.000} C_DIS
LIN {X -37.138,Y -37.308,Z -110.323,A -90.000,B 90.000,C 0.000} C_DIS
LIN {X -37.098,Y -37.308,Z -109.605,A -90.000,B 90.000,C 0.000} C_DIS
LIN {X -37.067,Y -37.308,Z -108.312,A -90.000,B 90.000,C 0.000} C_DIS
LIN {X -37.044,Y -37.308,Z -107.687,A -90.000,B 90.000,C 0.000} C_DIS
LIN {X -37.019,Y -37.308,Z -107.440,A -90.000,B 90.000,C 0.000} C_DIS
LIN {X -36.997,Y -37.308,Z -107.279,A -90.000,B 90.000,C 0.000} C_DIS
LIN {X -36.823,Y -37.308,Z -106.206,A -90.000,B 90.000,C 0.000} C_DIS
LIN {X -36.610,Y -37.308,Z -104.975,A -90.000,B 90.000,C 0.000} C_DIS
LIN {X -35.979,Y -37.308,Z -102.394,A -90.000,B 90.000,C 0.000} C_DIS
LIN {X -35.937,Y -37.308,Z -102.230,A -90.000,B 90.000,C 0.000} C_DIS
LIN {X -35.639,Y -37.308,Z -101.238,A -90.000,B 90.000,C 0.000} C_DIS
LIN {X -35.073,Y -37.308,Z -99.393,A -90.000,B 90.000,C 0.000} C_DIS
LIN {X -34.800,Y -37.308,Z -98.407,A -90.000,B 90.000,C 0.000} C_DIS
LIN {X -34.666,Y -37.308,Z -97.826,A -90.000,B 90.000,C 0.000} C_DIS
LIN {X -34.617,Y -37.308,Z -97.645,A -90.000,B 90.000,C 0.000} C_DIS
LIN {X -34.622,Y -37.308,Z -97.621,A -90.000,B 90.000,C 0.000} C_DIS
LIN {X -34.940,Y -37.308,Z -96.995,A -90.000,B 90.000,C 0.000} C_DIS
LIN {X -35.388,Y -37.308,Z -96.416,A -90.000,B 90.000,C 0.000} C_DIS
LIN {X -35.838,Y -37.308,Z -95.804,A -90.000,B 90.000,C 0.000} C_DIS
LIN {X -36.861,Y -37.308,Z -94.480,A -90.000,B 90.000,C 0.000} C_DIS
LIN {X -36.992,Y -37.308,Z -94.308,A -90.000,B 90.000,C 0.000} C_DIS
LIN {X -37.222,Y -37.308,Z -93.958,A -90.000,B 90.000,C 0.000} C_DIS
LIN {X -38.271,Y -37.308,Z -92.169,A -90.000,B 90.000,C 0.000} C_DIS
LIN {X -38.404,Y -37.308,Z -91.921,A -90.000,B 90.000,C 0.000} C_DIS
LIN {X -38.813,Y -37.308,Z -91.094,A -90.000,B 90.000,C 0.000} C_DIS
LIN {X -39.292,Y -37.308,Z -90.109,A -90.000,B 90.000,C 0.000} C_DIS
LIN {X -39.568,Y -37.308,Z -89.332,A -90.000,B 90.000,C 0.000} C_DIS
LIN {X -39.754,Y -37.308,Z -88.751,A -90.000,B 90.000,C 0.000} C_DIS
LIN {X -40.030,Y -37.308,Z -87.735,A -90.000,B 90.000,C 0.000} C_DIS
LIN {X -40.197,Y -37.308,Z -87.084,A -90.000,B 90.000,C 0.000} C_DIS
LIN {X -40.286,Y -37.308,Z -86.626,A -90.000,B 90.000,C 0.000} C_DIS
LIN {X -40.316,Y -37.308,Z -86.391,A -90.000,B 90.000,C 0.000} C_DIS
LIN {X -40.350,Y -37.308,Z -84.333,A -90.000,B 90.000,C 0.000} C_DIS
LIN {X -40.346,Y -37.308,Z -84.202,A -90.000,B 90.000,C 0.000} C_DIS
LIN {X -40.326,Y -37.308,Z -83.966,A -90.000,B 90.000,C 0.000} C_DIS
LIN {X -39.885,Y -37.308,Z -82.220,A -90.000,B 90.000,C 0.000} C_DIS
LIN {X -39.849,Y -37.308,Z -82.062,A -90.000,B 90.000,C 0.000} C_DIS
LIN {X -39.780,Y -37.308,Z -81.835,A -90.000,B 90.000,C 0.000} C_DIS
LIN {X -38.989,Y -37.308,Z -80.095,A -90.000,B 90.000,C 0.000} C_DIS
LIN {X -38.975,Y -37.308,Z -80.060,A -90.000,B 90.000,C 0.000} C_DIS
LIN {X -38.860,Y -37.308,Z -79.852,A -90.000,B 90.000,C 0.000} C_DIS
LIN {X -38.744,Y -37.308,Z -79.660,A -90.000,B 90.000,C 0.000} C_DIS
LIN {X -37.741,Y -37.308,Z -78.130,A -90.000,B 90.000,C 0.000} C_DIS
LIN {X -36.964,Y -37.308,Z -77.043,A -90.000,B 90.000,C 0.000} C_DIS
LIN {X -36.377,Y -37.308,Z -76.349,A -90.000,B 90.000,C 0.000} C_DIS
LIN {X -36.221,Y -37.308,Z -76.170,A -90.000,B 90.000,C 0.000} C_DIS
LIN {X -35.694,Y -37.308,Z -75.642,A -90.000,B 90.000,C 0.000} C_DIS
LIN {X -34.538,Y -37.308,Z -74.674,A -90.000,B 90.000,C 0.000} C_DIS
LIN {X -34.359,Y -37.308,Z -74.527,A -90.000,B 90.000,C 0.000} C_DIS
LIN {X -34.243,Y -37.308,Z -74.440,A -90.000,B 90.000,C 0.000} C_DIS
LIN {X -34.183,Y -37.308,Z -74.406,A -90.000,B 90.000,C 0.000} C_DIS
LIN {X -33.856,Y -37.308,Z -74.256,A -90.000,B 90.000,C 0.000} C_DIS
LIN {X -32.600,Y -37.308,Z -73.756,A -90.000,B 90.000,C 0.000} C_DIS
LIN {X -31.550,Y -37.308,Z -73.451,A -90.000,B 90.000,C 0.000} C_DIS
LIN {X -31.319,Y -37.308,Z -73.398,A -90.000,B 90.000,C 0.000} C_DIS
LIN {X -30.815,Y -37.308,Z -73.291,A -90.000,B 90.000,C 0.000} C_DIS
LIN {X -29.476,Y -37.308,Z -73.161,A -90.000,B 90.000,C 0.000} C_DIS
LIN {X -29.239,Y -37.308,Z -73.159,A -90.000,B 90.000,C 0.000} C_DIS
LIN {X -28.930,Y -37.308,Z -73.162,A -90.000,B 90.000,C 0.000} C_DIS
LIN {X -28.836,Y -37.308,Z -73.169,A -90.000,B 90.000,C 0.000} C_DIS
LIN {X -28.690,Y -37.308,Z -73.199,A -90.000,B 90.000,C 0.000} C_DIS
LIN {X -26.922,Y -37.308,Z -73.480,A -90.000,B 90.000,C 0.000} C_DIS
LIN {X -26.690,Y -37.308,Z -73.527,A -90.000,B 90.000,C 0.000} C_DIS
LIN {X -26.406,Y -37.308,Z -73.605,A -90.000,B 90.000,C 0.000} C_DIS
LIN {X -25.102,Y -37.308,Z -73.876,A -90.000,B 90.000,C 0.000} C_DIS
LIN {X -23.846,Y -37.308,Z -74.062,A -90.000,B 90.000,C 0.000} C_DIS
LIN {X -23.616,Y -37.308,Z -74.057,A -90.000,B 90.000,C 0.000} C_DIS
LIN {X -22.926,Y -37.308,Z -74.026,A -90.000,B 90.000,C 0.000} C_DIS
LIN {X -22.457,Y -37.308,Z -73.832,A -90.000,B 90.000,C 0.000} C_DIS
LIN {X -21.577,Y -37.308,Z -73.225,A -90.000,B 90.000,C 0.000} C_DIS
LIN {X -21.409,Y -37.308,Z -73.099,A -90.000,B 90.000,C 0.000} C_DIS
LIN {X -21.222,Y -37.308,Z -72.961,A -90.000,B 90.000,C 0.000} C_DIS
LIN {X -20.387,Y -37.308,Z -72.503,A -90.000,B 90.000,C 0.000} C_DIS
LIN {X -20.077,Y -37.308,Z -72.337,A -90.000,B 90.000,C 0.000} C_DIS
LIN {X -18.745,Y -37.308,Z -71.769,A -90.000,B 90.000,C 0.000} C_DIS
LIN {X -18.472,Y -37.308,Z -71.650,A -90.000,B 90.000,C 0.000} C_DIS
LIN {X -18.128,Y -37.308,Z -71.526,A -90.000,B 90.000,C 0.000} C_DIS
LIN {X -18.076,Y -37.308,Z -71.510,A -90.000,B 90.000,C 0.000} C_DIS
LIN {X -17.813,Y -37.308,Z -71.452,A -90.000,B 90.000,C 0.000} C_DIS
LIN {X -17.515,Y -37.308,Z -71.389,A -90.000,B 90.000,C 0.000} C_DIS
LIN {X -16.379,Y -37.308,Z -71.226,A -90.000,B 90.000,C 0.000} C_DIS
LIN {X -15.693,Y -37.308,Z -71.146,A -90.000,B 90.000,C 0.000} C_DIS
LIN {X -15.342,Y -37.308,Z -71.123,A -90.000,B 90.000,C 0.000} C_DIS
LIN {X -14.381,Y -37.308,Z -71.095,A -90.000,B 90.000,C 0.000} C_DIS
LIN {X -12.590,Y -37.308,Z -71.070,A -90.000,B 90.000,C 0.000} C_DIS
LIN {X -11.684,Y -37.308,Z -71.124,A -90.000,B 90.000,C 0.000} C_DIS
LIN {X -10.057,Y -37.308,Z -71.250,A -90.000,B 90.000,C 0.000} C_DIS
LIN {X -8.883,Y -37.308,Z -71.339,A -90.000,B 90.000,C 0.000} C_DIS
LIN {X -7.142,Y -37.308,Z -71.581,A -90.000,B 90.000,C 0.000} C_DIS
LIN {X -4.965,Y -37.308,Z -71.858,A -90.000,B 90.000,C 0.000} C_DIS
LIN {X -4.349,Y -37.308,Z -71.976,A -90.000,B 90.000,C 0.000} C_DIS
LIN {X -3.214,Y -37.308,Z -72.171,A -90.000,B 90.000,C 0.000} C_DIS
LIN {X -2.131,Y -37.308,Z -72.344,A -90.000,B 90.000,C 0.000} C_DIS
LIN {X -0.215,Y -37.308,Z -72.603,A -90.000,B 90.000,C 0.000} C_DIS
LIN {X 0.491,Y -37.308,Z -72.732,A -90.000,B 90.000,C 0.000} C_DIS
LIN {X 0.692,Y -37.308,Z -72.762,A -90.000,B 90.000,C 0.000} C_DIS
LIN {X 1.775,Y -37.308,Z -72.799,A -90.000,B 90.000,C 0.000} C_DIS
LIN {X 2.414,Y -37.308,Z -72.785,A -90.000,B 90.000,C 0.000} C_DIS
LIN {X 2.642,Y -37.308,Z -72.723,A -90.000,B 90.000,C 0.000} C_DIS
LIN {X 3.221,Y -37.308,Z -72.505,A -90.000,B 90.000,C 0.000} C_DIS
LIN {X 3.607,Y -37.308,Z -72.078,A -90.000,B 90.000,C 0.000} C_DIS
LIN {X 3.765,Y -37.308,Z -71.865,A -90.000,B 90.000,C 0.000} C_DIS
LIN {X 4.154,Y -37.308,Z -71.285,A -90.000,B 90.000,C 0.000} C_DIS
LIN {X 4.279,Y -37.308,Z -71.157,A -90.000,B 90.000,C 0.000} C_DIS
LIN {X 4.382,Y -37.308,Z -71.056,A -90.000,B 90.000,C 0.000} C_DIS
LIN {X 4.572,Y -37.308,Z -70.914,A -90.000,B 90.000,C 0.000} C_DIS
LIN {X 4.855,Y -37.308,Z -70.728,A -90.000,B 90.000,C 0.000} C_DIS
LIN {X 5.532,Y -37.308,Z -70.237,A -90.000,B 90.000,C 0.000} C_DIS
LIN {X 5.747,Y -37.308,Z -70.138,A -90.000,B 90.000,C 0.000} C_DIS
LIN {X 7.163,Y -37.308,Z -69.625,A -90.000,B 90.000,C 0.000} C_DIS
LIN {X 7.377,Y -37.308,Z -69.552,A -90.000,B 90.000,C 0.000} C_DIS
LIN {X 7.517,Y -37.308,Z -69.510,A -90.000,B 90.000,C 0.000} C_DIS
LIN {X 7.707,Y -37.308,Z -69.468,A -90.000,B 90.000,C 0.000} C_DIS
LIN {X 8.293,Y -37.308,Z -69.343,A -90.000,B 90.000,C 0.000} C_DIS
LIN {X 9.928,Y -37.308,Z -69.155,A -90.000,B 90.000,C 0.000} C_DIS
LIN {X 10.209,Y -37.308,Z -69.173,A -90.000,B 90.000,C 0.000} C_DIS
LIN {X 11.122,Y -37.308,Z -69.271,A -90.000,B 90.000,C 0.000} C_DIS
LIN {X 11.891,Y -37.308,Z -69.325,A -90.000,B 90.000,C 0.000} C_DIS
LIN {X 12.280,Y -37.308,Z -69.401,A -90.000,B 90.000,C 0.000} C_DIS
LIN {X 13.067,Y -37.308,Z -69.564,A -90.000,B 90.000,C 0.000} C_DIS
LIN {X 13.368,Y -37.308,Z -69.623,A -90.000,B 90.000,C 0.000} C_DIS
LIN {X 13.404,Y -37.308,Z -69.626,A -90.000,B 90.000,C 0.000} C_DIS
LIN {X 13.413,Y -37.308,Z -69.554,A -90.000,B 90.000,C 0.000} C_DIS
LIN {X 13.440,Y -37.308,Z -69.302,A -90.000,B 90.000,C 0.000} C_DIS
LIN {X 13.480,Y -37.308,Z -69.004,A -90.000,B 90.000,C 0.000} C_DIS
LIN {X 13.543,Y -37.308,Z -68.647,A -90.000,B 90.000,C 0.000} C_DIS
LIN {X 13.665,Y -37.308,Z -68.265,A -90.000,B 90.000,C 0.000} C_DIS
LIN {X 13.686,Y -37.308,Z -68.205,A -90.000,B 90.000,C 0.000} C_DIS
LIN {X 13.760,Y -37.308,Z -68.013,A -90.000,B 90.000,C 0.000} C_DIS
LIN {X 13.826,Y -37.308,Z -67.871,A -90.000,B 90.000,C 0.000} C_DIS
LIN {X 13.927,Y -37.308,Z -67.691,A -90.000,B 90.000,C 0.000} C_DIS
LIN {X 14.012,Y -37.308,Z -67.559,A -90.000,B 90.000,C 0.000} C_DIS
LIN {X 14.324,Y -37.308,Z -67.130,A -90.000,B 90.000,C 0.000} C_DIS
LIN {X 14.658,Y -37.308,Z -66.734,A -90.000,B 90.000,C 0.000} C_DIS
LIN {X 14.936,Y -37.308,Z -66.482,A -90.000,B 90.000,C 0.000} C_DIS
LIN {X 15.247,Y -37.308,Z -66.267,A -90.000,B 90.000,C 0.000} C_DIS
LIN {X 15.561,Y -37.308,Z -66.105,A -90.000,B 90.000,C 0.000} C_DIS
LIN {X 15.585,Y -37.308,Z -66.094,A -90.000,B 90.000,C 0.000} C_DIS
LIN {X 15.942,Y -37.308,Z -65.967,A -90.000,B 90.000,C 0.000} C_DIS
LIN {X 16.313,Y -37.308,Z -65.889,A -90.000,B 90.000,C 0.000} C_DIS
LIN {X 16.331,Y -37.308,Z -65.886,A -90.000,B 90.000,C 0.000} C_DIS
LIN {X 16.941,Y -37.308,Z -65.758,A -90.000,B 90.000,C 0.000} C_DIS
LIN {X 17.316,Y -37.308,Z -65.730,A -90.000,B 90.000,C 0.000} C_DIS
LIN {X 17.711,Y -37.308,Z -65.750,A -90.000,B 90.000,C 0.000} C_DIS
LIN {X 18.083,Y -37.308,Z -65.820,A -90.000,B 90.000,C 0.000} C_DIS
LIN {X 18.673,Y -37.308,Z -65.936,A -90.000,B 90.000,C 0.000} C_DIS
LIN {X 18.853,Y -37.308,Z -65.976,A -90.000,B 90.000,C 0.000} C_DIS
LIN {X 19.146,Y -37.308,Z -66.066,A -90.000,B 90.000,C 0.000} C_DIS
LIN {X 19.149,Y -37.308,Z -66.062,A -90.000,B 90.000,C 0.000} C_DIS
LIN {X 19.421,Y -37.308,Z -65.641,A -90.000,B 90.000,C 0.000} C_DIS
LIN {X 19.588,Y -37.308,Z -65.426,A -90.000,B 90.000,C 0.000} C_DIS
LIN {X 19.652,Y -37.308,Z -65.350,A -90.000,B 90.000,C 0.000} C_DIS
LIN {X 19.837,Y -37.308,Z -65.168,A -90.000,B 90.000,C 0.000} C_DIS
LIN {X 19.910,Y -37.308,Z -65.102,A -90.000,B 90.000,C 0.000} C_DIS
LIN {X 20.120,Y -37.308,Z -64.948,A -90.000,B 90.000,C 0.000} C_DIS
LIN {X 20.201,Y -37.308,Z -64.892,A -90.000,B 90.000,C 0.000} C_DIS
LIN {X 20.430,Y -37.308,Z -64.769,A -90.000,B 90.000,C 0.000} C_DIS
LIN {X 20.518,Y -37.308,Z -64.724,A -90.000,B 90.000,C 0.000} C_DIS
LIN {X 20.855,Y -37.308,Z -64.602,A -90.000,B 90.000,C 0.000} C_DIS
LIN {X 21.323,Y -37.308,Z -64.503,A -90.000,B 90.000,C 0.000} C_DIS
LIN {X 21.857,Y -37.308,Z -64.461,A -90.000,B 90.000,C 0.000} C_DIS
LIN {X 22.235,Y -37.308,Z -64.482,A -90.000,B 90.000,C 0.000} C_DIS
LIN {X 22.826,Y -37.308,Z -64.572,A -90.000,B 90.000,C 0.000} C_DIS
LIN {X 23.214,Y -37.308,Z -64.679,A -90.000,B 90.000,C 0.000} C_DIS
LIN {X 23.311,Y -37.308,Z -64.714,A -90.000,B 90.000,C 0.000} C_DIS
LIN {X 23.930,Y -37.308,Z -64.945,A -90.000,B 90.000,C 0.000} C_DIS
LIN {X 24.026,Y -37.308,Z -64.991,A -90.000,B 90.000,C 0.000} C_DIS
LIN {X 24.283,Y -37.308,Z -64.854,A -90.000,B 90.000,C 0.000} C_DIS
LIN {X 24.465,Y -37.308,Z -64.787,A -90.000,B 90.000,C 0.000} C_DIS
LIN {X 24.571,Y -37.308,Z -64.741,A -90.000,B 90.000,C 0.000} C_DIS
LIN {X 24.913,Y -37.308,Z -64.619,A -90.000,B 90.000,C 0.000} C_DIS
LIN {X 24.974,Y -37.308,Z -64.600,A -90.000,B 90.000,C 0.000} C_DIS
LIN {X 25.183,Y -37.308,Z -64.518,A -90.000,B 90.000,C 0.000} C_DIS
LIN {X 25.280,Y -37.308,Z -64.473,A -90.000,B 90.000,C 0.000} C_DIS
LIN {X 25.379,Y -37.308,Z -64.416,A -90.000,B 90.000,C 0.000} C_DIS
LIN {X 25.496,Y -37.308,Z -64.347,A -90.000,B 90.000,C 0.000} C_DIS
LIN {X 25.566,Y -37.308,Z -64.301,A -90.000,B 90.000,C 0.000} C_DIS
LIN {X 25.681,Y -37.308,Z -64.213,A -90.000,B 90.000,C 0.000} C_DIS
LIN {X 25.784,Y -37.308,Z -64.129,A -90.000,B 90.000,C 0.000} C_DIS
LIN {X 25.891,Y -37.308,Z -64.028,A -90.000,B 90.000,C 0.000} C_DIS
LIN {X 26.039,Y -37.308,Z -63.863,A -90.000,B 90.000,C 0.000} C_DIS
LIN {X 26.318,Y -37.308,Z -63.532,A -90.000,B 90.000,C 0.000} C_DIS
LIN {X 26.359,Y -37.308,Z -63.492,A -90.000,B 90.000,C 0.000} C_DIS
LIN {X 26.420,Y -37.308,Z -63.418,A -90.000,B 90.000,C 0.000} C_DIS
LIN {X 26.670,Y -37.308,Z -63.172,A -90.000,B 90.000,C 0.000} C_DIS
LIN {X 26.954,Y -37.308,Z -62.964,A -90.000,B 90.000,C 0.000} C_DIS
LIN {X 27.264,Y -37.308,Z -62.798,A -90.000,B 90.000,C 0.000} C_DIS
LIN {X 27.432,Y -37.308,Z -62.736,A -90.000,B 90.000,C 0.000} C_DIS
LIN {X 27.376,Y -37.308,Z -62.251,A -90.000,B 90.000,C 0.000} C_DIS
LIN {X 27.270,Y -37.308,Z -61.182,A -90.000,B 90.000,C 0.000} C_DIS
LIN {X 27.245,Y -37.308,Z -60.443,A -90.000,B 90.000,C 0.000} C_DIS
LIN {X 27.244,Y -37.308,Z -60.364,A -90.000,B 90.000,C 0.000} C_DIS
LIN {X 27.251,Y -37.308,Z -59.869,A -90.000,B 90.000,C 0.000} C_DIS
LIN {X 27.314,Y -37.308,Z -59.294,A -90.000,B 90.000,C 0.000} C_DIS
LIN {X 27.374,Y -37.308,Z -58.858,A -90.000,B 90.000,C 0.000} C_DIS
LIN {X 27.470,Y -37.308,Z -58.469,A -90.000,B 90.000,C 0.000} C_DIS
LIN {X 27.575,Y -37.308,Z -58.057,A -90.000,B 90.000,C 0.000} C_DIS
LIN {X 27.736,Y -37.308,Z -57.639,A -90.000,B 90.000,C 0.000} C_DIS
